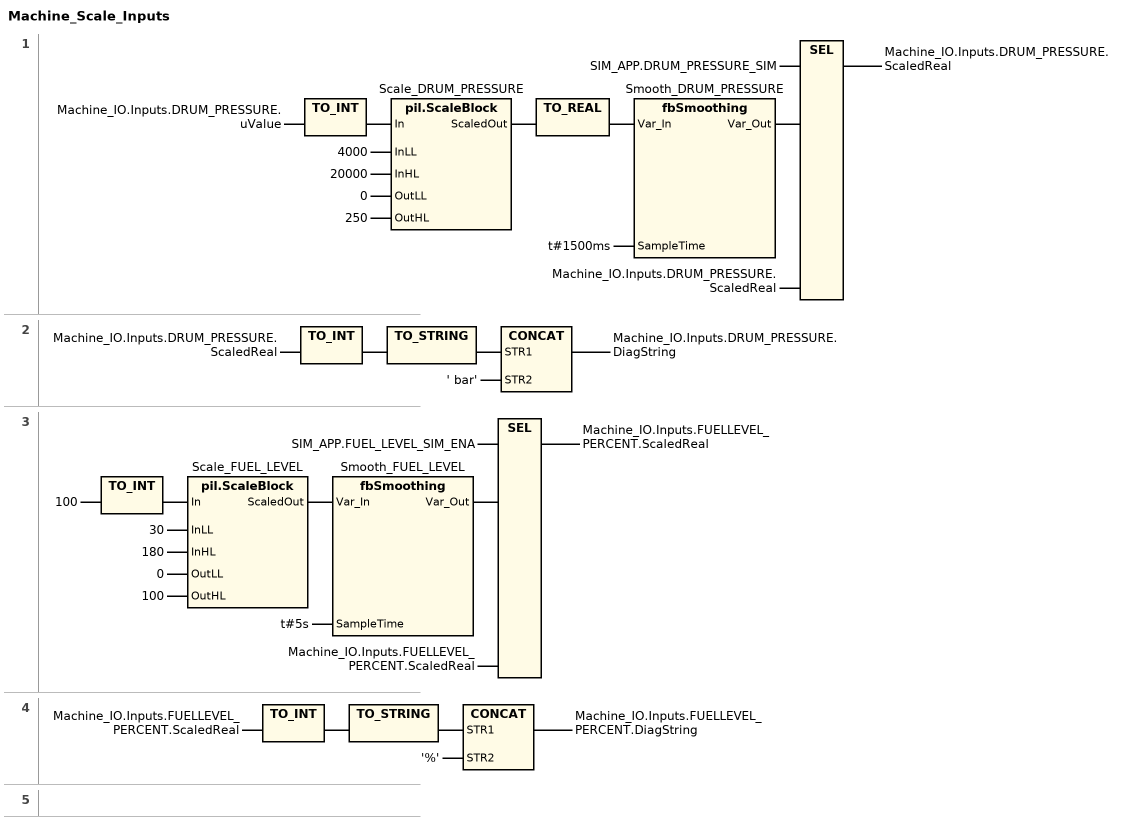
// NETWORK 1
Scale_DRUM_PRESSURE(
    In := TO_INT(Machine_IO.Inputs.DRUM_PRESSURE.uValue),
    InLL := 4000,
    InHL := 20000,
    OutLL := 0,
    OutHL := 250); // pil.ScaleBlock
Smooth_DRUM_PRESSURE(Var_In := TO_REAL(Scale_DRUM_PRESSURE.ScaledOut), SampleTime := t#1500ms); // fbSmoothing
Machine_IO.Inputs.DRUM_PRESSURE.ScaledReal := SEL(SIM_APP.DRUM_PRESSURE_SIM, Smooth_DRUM_PRESSURE.Var_Out, Machine_IO.Inputs.DRUM_PRESSURE.ScaledReal);

// NETWORK 2
Machine_IO.Inputs.DRUM_PRESSURE.DiagString := CONCAT(STR1 := TO_STRING(TO_INT(Machine_IO.Inputs.DRUM_PRESSURE.ScaledReal)), STR2 := ' bar');

// NETWORK 3
Scale_FUEL_LEVEL(In := TO_INT(100), InLL := 30, InHL := 180, OutLL := 0, OutHL := 100); // pil.ScaleBlock
Smooth_FUEL_LEVEL(Var_In := Scale_FUEL_LEVEL.ScaledOut, SampleTime := t#5s); // fbSmoothing
Machine_IO.Inputs.FUELLEVEL_PERCENT.ScaledReal := SEL(SIM_APP.FUEL_LEVEL_SIM_ENA, Smooth_FUEL_LEVEL.Var_Out, Machine_IO.Inputs.FUELLEVEL_PERCENT.ScaledReal);

// NETWORK 4
Machine_IO.Inputs.FUELLEVEL_PERCENT.DiagString := CONCAT(STR1 := TO_STRING(TO_INT(Machine_IO.Inputs.FUELLEVEL_PERCENT.ScaledReal)), STR2 := '%');

// NETWORK 5

END_PROGRAM

// Device/Application/App_PLC/fbSmoothing
FUNCTION_BLOCK fbSmoothing
VAR_INPUT
	Var_In: REAL;
	SampleTime: TIME;
END_VAR
VAR_OUTPUT
	Var_Out: REAL;
END_VAR
VAR
	Timer: TON;
	SampleArray: ARRAY [0..49] OF REAL;
	ArraySampleTime: TIME;
	Timer2: TON;
END_VAR

ArraySampleTime:= SampleTime/50;
Timer(IN:=NOT Timer.Q, PT:=ArraySampleTime, Q=>, ET=> );

IF Timer.Q=TRUE THEN

SampleArray[49]:=SampleArray[48];
SampleArray[48]:=SampleArray[47];
SampleArray[47]:=SampleArray[46];
SampleArray[46]:=SampleArray[45];
SampleArray[45]:=SampleArray[44];
SampleArray[44]:=SampleArray[43];
SampleArray[43]:=SampleArray[42];
SampleArray[42]:=SampleArray[41];
SampleArray[41]:=SampleArray[40];
SampleArray[40]:=SampleArray[39];
SampleArray[39]:=SampleArray[38];
SampleArray[38]:=SampleArray[37];
SampleArray[37]:=SampleArray[36];
SampleArray[36]:=SampleArray[35];
SampleArray[35]:=SampleArray[34];
SampleArray[34]:=SampleArray[33];
SampleArray[33]:=SampleArray[32];
SampleArray[32]:=SampleArray[31];
SampleArray[31]:=SampleArray[30];
SampleArray[30]:=SampleArray[29];
SampleArray[29]:=SampleArray[28];
SampleArray[28]:=SampleArray[27];
SampleArray[27]:=SampleArray[26];
SampleArray[26]:=SampleArray[25];
SampleArray[25]:=SampleArray[24];
SampleArray[24]:=SampleArray[23];
SampleArray[23]:=SampleArray[22];
SampleArray[22]:=SampleArray[21];
SampleArray[21]:=SampleArray[20];
SampleArray[20]:=SampleArray[19];
SampleArray[19]:=SampleArray[18];
SampleArray[18]:=SampleArray[17];
SampleArray[17]:=SampleArray[16];
SampleArray[16]:=SampleArray[15];
SampleArray[15]:=SampleArray[14];
SampleArray[14]:=SampleArray[13];
SampleArray[13]:=SampleArray[12];
SampleArray[12]:=SampleArray[11];
SampleArray[11]:=SampleArray[10];
SampleArray[10]:=SampleArray[9];
SampleArray[9]:=SampleArray[8];
SampleArray[8]:=SampleArray[7];
SampleArray[7]:=SampleArray[6];
SampleArray[6]:=SampleArray[5];
SampleArray[5]:=SampleArray[4];
SampleArray[4]:=SampleArray[3];
SampleArray[3]:=SampleArray[2];
SampleArray[2]:=SampleArray[1];
SampleArray[1]:=SampleArray[0];
SampleArray[0]:=Var_In;
END_IF

Timer2(IN:=NOT Timer2.Q, PT:=SampleTime, Q=>, ET=> );

IF Timer2.Q=TRUE THEN
Var_Out:= (
SampleArray[49] + SampleArray[48] + SampleArray[47] + SampleArray[46] + SampleArray[45] + SampleArray[44] + SampleArray[43] + SampleArray[42] + SampleArray[41] +SampleArray[40] +
SampleArray[39] + SampleArray[38] + SampleArray[37] + SampleArray[36] + SampleArray[35] + SampleArray[34] + SampleArray[33] + SampleArray[32] + SampleArray[31] +SampleArray[30] +
SampleArray[29] + SampleArray[28] + SampleArray[27] + SampleArray[26] + SampleArray[25] + SampleArray[24] + SampleArray[23] + SampleArray[22] + SampleArray[21] +SampleArray[20] +
SampleArray[19] + SampleArray[18] + SampleArray[17] + SampleArray[16] + SampleArray[15] + SampleArray[14] + SampleArray[13] + SampleArray[12] + SampleArray[11] +SampleArray[10] +
SampleArray[9] + SampleArray[8] + SampleArray[7] + SampleArray[6] + SampleArray[5] + SampleArray[4] + SampleArray[3] + SampleArray[2] + SampleArray[1] +SampleArray[0]
			)/50;
END_IF

END_FUNCTION_BLOCK

// Device/Application/LIBS/Logging/Log_File_Append
FUNCTION Log_File_Append : INT
VAR_INPUT
	LogString: STRING;
	szFileName : STRING;		
	Updated_Flag: REFERENCE TO INT;
END_VAR
VAR	
	hFile : RTS_IEC_HANDLE := RTS_INVALID_HANDLE;
	
	udiWriteError : RTS_IEC_RESULT;
	udiOpenError : RTS_IEC_RESULT;
	udiCloseError : RTS_IEC_RESULT;
	udiWrite : __XWORD;
	
	TempString: STRING;
	
	High_Res_millis: INT:=0;
	High_Res_Timestamp:	SYSTIME;
	High_Res_Timestamp_Result: RTS_IEC_RESULT;
	High_Res_Timestamp_DT: DT;
	High_Res_Timestamp_String: STRING;
END_VAR

// get the high res time stamp that has milliseconds
High_Res_Timestamp_Result:=SysTimeRtc.SysTimeRtcHighResGet(High_Res_Timestamp);

IF High_Res_Timestamp_Result <> CmpErrors.Errors.ERR_OK THEN
	Log_File_Append:=-1;
	RETURN;	
END_IF

High_Res_Timestamp_DT := TO_DT(High_Res_Timestamp/1000);
High_Res_millis := TO_INT(High_Res_Timestamp MOD 1000);

High_Res_Timestamp_String := OSCAT_BASIC.DT_TO_STRF(DTI:=High_Res_Timestamp_DT, MS:=High_Res_millis, FMT:='#N:#R:#T.#V,#H-#D-#A',LANG:=OSCAT_BASIC.language.DEFAULT);

hFile := SysFileOpen(szFile:=szFileName, am:=SysFile.AM_APPEND_PLUS, pResult:=ADR(udiOpenError));

IF hFile <> RTS_INVALID_HANDLE	THEN
	TempString:=CONCAT(TempString,LogString);	
	TempString:=CONCAT(TempString,',');
	TempString:=CONCAT(TempString,High_Res_Timestamp_String);	
	TempString:=CONCAT(TempString,'$0d$0a');
	udiWrite := SysFileWrite(hFile:=hFile, pbyBuffer:=ADR(TempString), ulSize:=INT_TO_UDINT(LEN(TempString)), pResult:=ADR(udiWriteError));

	udiCloseError  := SysFileClose(hFile:=hFile);
	Log_File_Append:=0;
	Updated_Flag:=Updated_Flag+1;
	RETURN;
END_IF

Log_File_Append:=-2;
RETURN;

END_FUNCTION

// Device/Application/App_Common/System/PLC_LOGGING
PROGRAM PLC_LOGGING
VAR
	Main_Log_Update: BOOL;
	Main_Log_Update_Reset_TON: TON;
	
	LOG_LINES: ARRAY [0..9] OF STRING(200);
	Log_File_Read_Lines_Check_FB: Log_File_Read_Lines;
	Log_File_Read_Lines_FB: Log_File_Read_Lines;
	MaxLines: INT :=10;
	
	Offset: INT;
	Number_Lines: INT;
END_VAR
VAR // added by the converter: edge detectors and wires of the graphical bodies
    _rt1, _rt2, _rt3, _rt4, _rt5 : R_TRIG;
    _w1, _w2, _w3 : BOOL;
END_VAR

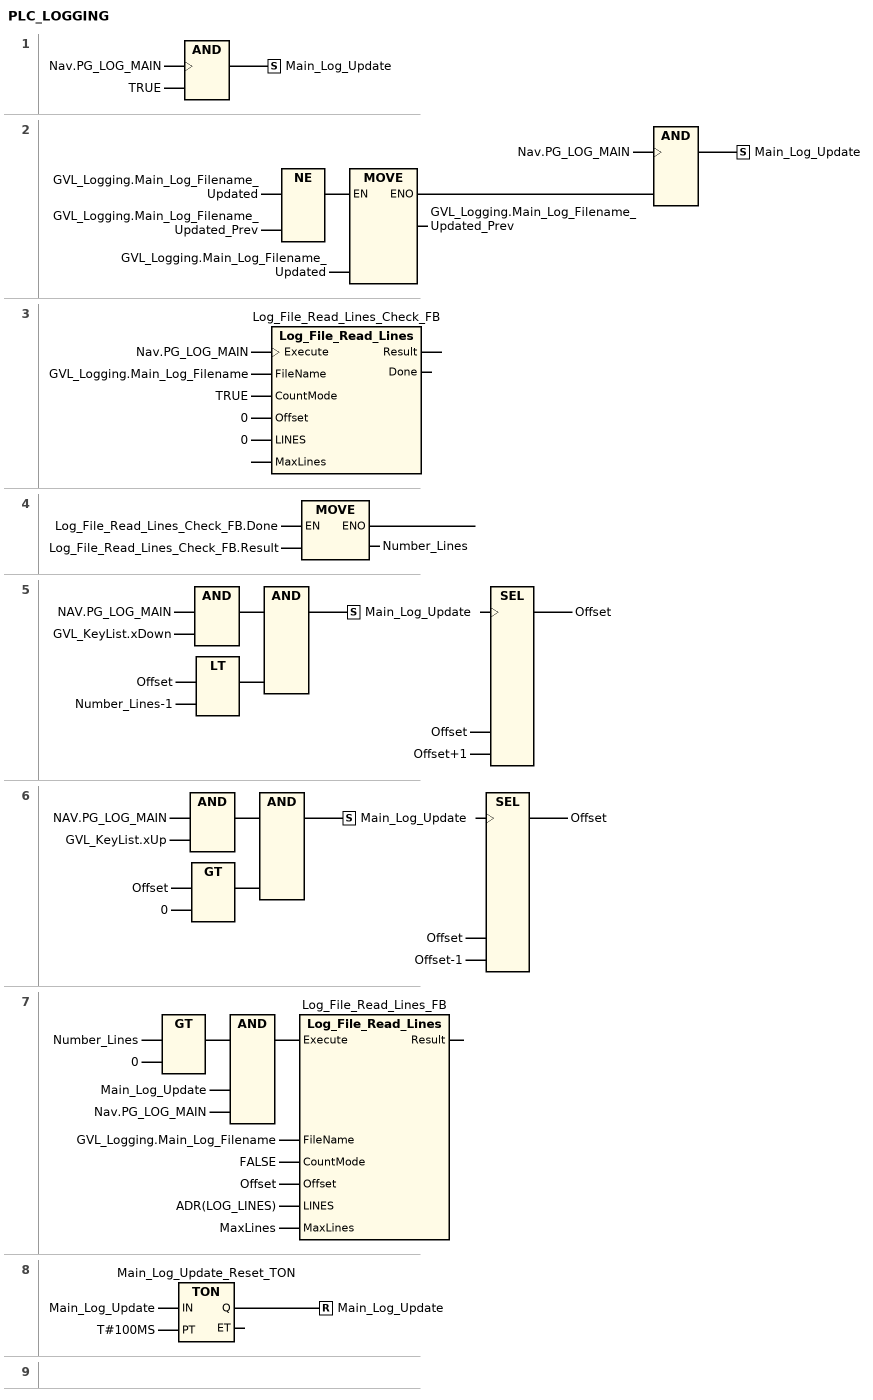
// NETWORK 1
_rt1(CLK := Nav.PG_LOG_MAIN);
Main_Log_Update S= _rt1.Q AND TRUE;

// NETWORK 2
_rt2(CLK := Nav.PG_LOG_MAIN);
_w1 := GVL_Logging.Main_Log_Filename_Updated <> GVL_Logging.Main_Log_Filename_Updated_Prev;
IF _w1 THEN GVL_Logging.Main_Log_Filename_Updated_Prev := GVL_Logging.Main_Log_Filename_Updated; END_IF
Main_Log_Update S= _rt2.Q AND _w1;

// NETWORK 3
_rt3(CLK := Nav.PG_LOG_MAIN);
Log_File_Read_Lines_Check_FB(
    Execute := _rt3.Q,
    FileName := GVL_Logging.Main_Log_Filename,
    CountMode := TRUE,
    Offset := 0,
    LINES := 0); // Log_File_Read_Lines

// NETWORK 4
IF Log_File_Read_Lines_Check_FB.Done THEN Number_Lines := Log_File_Read_Lines_Check_FB.Result; END_IF

// NETWORK 5
_w2 := (NAV.PG_LOG_MAIN AND GVL_KeyList.xDown) AND Offset < (Number_Lines-1);
Main_Log_Update S= _w2;
_rt4(CLK := _w2);
Offset := SEL(_rt4.Q, Offset, Offset+1);

// NETWORK 6
_w3 := (NAV.PG_LOG_MAIN AND GVL_KeyList.xUp) AND Offset > 0;
Main_Log_Update S= _w3;
_rt5(CLK := _w3);
Offset := SEL(_rt5.Q, Offset, Offset-1);

// NETWORK 7
Log_File_Read_Lines_FB(
    Execute := Number_Lines > 0 AND Main_Log_Update AND Nav.PG_LOG_MAIN,
    FileName := GVL_Logging.Main_Log_Filename,
    CountMode := FALSE,
    Offset := Offset,
    LINES := ADR(LOG_LINES),
    MaxLines := MaxLines); // Log_File_Read_Lines

// NETWORK 8
Main_Log_Update_Reset_TON(IN := Main_Log_Update, PT := T#100MS); // TON
Main_Log_Update R= Main_Log_Update_Reset_TON.Q;

// NETWORK 9

END_PROGRAM

// Device/Application/LIBS/Logging/Log_File_Read_Lines
FUNCTION_BLOCK Log_File_Read_Lines
VAR_INPUT
	Execute: BOOL;
	FileName: STRING;
	CountMode: BOOL;
	Offset: INT:=0;
	LINES: POINTER TO STRING(200);	
	MaxLines: INT:=10;
END_VAR
VAR	
	hFile : RTS_IEC_HANDLE := RTS_INVALID_HANDLE;
	
	udiReadError : RTS_IEC_RESULT;
	udiOpenError : RTS_IEC_RESULT;
	udiCloseError : RTS_IEC_RESULT;
	udiWrite : __XWORD;
	ReadSize : __XWORD;
	
	TempString: STRING(2);
	LineBuffer: STRING(200);
	
	NumLines:INT:=0;
	line_counter:INT :=0;

	op_index:INT :=0;
	dummy: INT;
	Finished:BOOL:=FALSE;
END_VAR

VAR_OUTPUT
	Result:INT;
	Done: BOOL;
END_VAR

IF Execute = FALSE THEN
	Result:=0;
	Done:=0;
	RETURN;
END_IF

IF MaxLines = 0 THEN
	RETURN;
END_IF

IF LINES <> 0 THEN
	FOR line_counter := 0 TO (MaxLines-1) BY 1 DO
		LINES[line_counter]:='';
	END_FOR;	
END_IF

IF CountMode = FALSE AND LINES = 0 THEN
	Result:= -1;
	RETURN;
END_IF

hFile := SysFileOpen(szFile:=FileName, am:=SysFile.AM_READ, pResult:=ADR(udiOpenError));

IF hFile = RTS_INVALID_HANDLE THEN
	Result:=-2;
	RETURN;	
END_IF

Finished := FALSE;

line_counter:=0;
LineBuffer:='';

WHILE Finished = FALSE DO
	ReadSize := SysFileRead(hFile:=hFile, pbyBuffer:=ADR(TempString), ulSize:=1, pResult:=ADR(udiReadError));
	
	IF ReadSize<= 0 THEN
		Finished:=TRUE;
	END_IF
	
	TempString:=LEFT(TempString,1);
	IF(TempString='$0D') THEN
		op_index:=line_counter-Offset;	
		IF op_index >= 0 AND op_index < (MaxLines-1) THEN
			IF CountMode = FALSE AND op_index < MaxLines AND (LEN(LineBuffer)>0) THEN
				IF LINES <> 0 THEN
					LINES[op_index]:='[';
					LINES[op_index]:=CONCAT(LINES[op_index],TO_STRING(line_counter));
					LINES[op_index]:=CONCAT(LINES[op_index],'] ');
					LINES[op_index]:=CONCAT(LINES[op_index],LineBuffer);				
				END_IF
			END_IF			
		END_IF
		line_counter:=line_counter+1;		
		LineBuffer:='';		
		
	ELSIF(TempString='$0A') THEN
		dummy:=dummy+1;
	ELSE
		LineBuffer:=CONCAT(LineBuffer,TempString);
	END_IF
END_WHILE

udiCloseError  := SysFileClose(hFile:=hFile);
Result:=line_counter;
Done:=1;
RETURN;

END_FUNCTION_BLOCK

// Device/Application/LIBS/Alarms/Functions/Alarm_Table_Main
PROGRAM Alarm_Table_Main
VAR CONSTANT
	NUM_LINES: WORD:=5;
END_VAR

VAR
	BASE_INDEX:WORD:=0;
	Lines: ARRAY [0..(NUM_LINES-1)] OF Alarm_Logger_Line_FB;
	INDEXS: ARRAY [0..(NUM_LINES-1)] OF WORD;
	X:WORD;
END_VAR

VAR_INPUT
	LIST: REFERENCE TO SLL_LOGGER_MAIN_SRUCT;
	NAV_UP: BOOL;
	NAV_DOWN: BOOL;
END_VAR


FOR X:= 0 TO (NUM_LINES-1) DO
	INDEXS[X]:=(BASE_INDEX+X) MOD LIST.LOGGER_LIST_SIZE;	
	Lines[X](INDEX:=INDEXS[X],ITEM:=LIST.LOGGER_LIST[INDEXS[X]]);
END_FOR

IF NAV_UP THEN
	IF BASE_INDEX > 0 THEN 
		BASE_INDEX:=BASE_INDEX-1;
	ELSE
		BASE_INDEX:= LIST.LOGGER_LIST_SIZE-1;
	END_IF
END_IF

IF NAV_DOWN THEN
	IF BASE_INDEX <  (LIST.LOGGER_LIST_SIZE-2) THEN 
		BASE_INDEX:=BASE_INDEX+1;
	ELSE
		BASE_INDEX:= 0;
	END_IF
END_IF

END_PROGRAM

// Device/Application/LIBS/Alarms/Functions/Alarm_Logger_Line_FB
FUNCTION_BLOCK Alarm_Logger_Line_FB
VAR_INPUT
	INDEX: WORD;
	ITEM: REFERENCE TO SLL_LOGGER_ITEM;
END_VAR
VAR_OUTPUT
	oIndex:STRING;
	oID:STRING;
	oDescription: STRING;
	oTime: STRING;
	oAdd_Info: STRING;
	oSquareColour: DWORD;
END_VAR
VAR
	InitDone:BOOL :=FALSE;
	TempString: STRING;
	
	High_Res_millis: INT:=0;
	High_Res_Timestamp:	SYSTIME;
	High_Res_Timestamp_DT: DT;
END_VAR


oIndex:='[';
oIndex:=CONCAT(oIndex,TO_STRING(INDEX));
oIndex:=CONCAT(oIndex,']');

IF ITEM.ID > 0 THEN
	oID:=CONCAT('ID:',TO_STRING(ITEM.ID));	
	IF ITEM.Group.ErrorIO OR ITEM.Group.WarningIO THEN
		TempString := Alarm_ID_GetText('AlarmGroup_IO',TO_STRING(ITEM.ID));
	END_IF

	IF ITEM.Group.ErrorApp OR ITEM.Group.WarningApp THEN
		TempString := Alarm_ID_GetText('AlarmGroup_App',TO_STRING(ITEM.ID));
	END_IF
		

	IF TempString = '' THEN
		oDescription:=TO_STRING(ITEM.ID);
	END_IF;
	
	oDescription:=TempString;
	
	High_Res_Timestamp:=ITEM.TimeDateTriggered;
	High_Res_Timestamp_DT := TO_DT(High_Res_Timestamp/1000);
	High_Res_millis := TO_INT(High_Res_Timestamp MOD 1000);
	IF GVL_System.USA_Time_Format THEN
		oTime:= OSCAT_BASIC.DT_TO_STRF(DTI:=High_Res_Timestamp_DT, MS:=High_Res_millis, FMT:='#N:#R:#T.#V,#D-#H-#A',LANG:=OSCAT_BASIC.language.DEFAULT);
	ELSE
		oTime:= OSCAT_BASIC.DT_TO_STRF(DTI:=High_Res_Timestamp_DT, MS:=High_Res_millis, FMT:='#N:#R:#T.#V,#H-#D-#A',LANG:=OSCAT_BASIC.language.DEFAULT);
	END_IF

	oAdd_Info:=ITEM.Addtional_Info;
	
	IF ITEM.Flags.Active THEN
		oSquareColour:=GVL_Viz.Alarm_Log_Active_Colour;
	ELSE
		oSquareColour:=GVL_Viz.Alarm_Log_InActive_Colour;
	END_IF
ELSE
	oID:='';
	oDescription:='';
	oTime:='';
	oAdd_Info:='';
	oSquareColour:=GVL_Viz.Alarm_Log_None_Colour;
END_IF

END_FUNCTION_BLOCK

// Device/Application/LIBS/Alarms/Functions/Alarm_ID_GetText
FUNCTION Alarm_ID_GetText : STRING
VAR_INPUT
	TextListName: STRING;
	ItemName:STRING;	
END_VAR
VAR
	Current : STRING:='';
	TextListItem:STRING:='';
END_VAR

Current := DynamicTextGetCurrentLanguage();

IF Current = '' THEN
	TextListItem:=DynamicTextGetDefaultText(ADR(TextListName), ADR(ItemName))^;
ELSE
	TextListItem:=DynamicTextGetText(ADR(TextListName), ADR(ItemName))^;
END_IF

Alarm_ID_GetText:=TextListItem;

END_FUNCTION

// Device/Application/LIBS/Alarms/Functions/Alarm_Log_Clear_ALL
FUNCTION Alarm_Log_Clear_ALL : INT
VAR_INPUT
	LIST: REFERENCE TO SLL_LOGGER_MAIN_SRUCT;
	ENA: BOOL;
END_VAR
VAR_OUTPUT
END_VAR
VAR
	X:WORD;
	Empty_ITEM:SLL_LOGGER_ITEM;
END_VAR

IF ENA = FALSE THEN
	RETURN;	
END_IF

FOR X :=0 TO (LIST.LOGGER_LIST_SIZE-1) BY 1 DO
	LIST.LOGGER_LIST[X]:=Empty_ITEM;
END_FOR

END_FUNCTION

// Device/Application/LIBS/Alarms/Functions/Alarm_Log_Clear_ALL_Inactive
FUNCTION Alarm_Log_Clear_ALL_Inactive : INT
VAR_INPUT
	LIST: REFERENCE TO SLL_LOGGER_MAIN_SRUCT;
	ENA: BOOL;
END_VAR
VAR_OUTPUT
END_VAR
VAR
	X:WORD;
	Z:WORD;
	Empty_ITEM:SLL_LOGGER_ITEM;
END_VAR

IF ENA = FALSE THEN
	RETURN;	
END_IF

FOR X :=0 TO (LIST.LOGGER_LIST_SIZE-1) BY 1 DO
	IF LIST.LOGGER_LIST[X].ID > 0 THEN
		// got a id of some sort...
		IF LIST.LOGGER_LIST[X].Flags.Active = FALSE THEN
			// wipe this record 
			LIST.LOGGER_LIST[X]:=Empty_ITEM;
	
			// loose this record..shift up the date towards the start!
			FOR Z:= X TO (LIST.LOGGER_LIST_SIZE-2) BY 1 DO
				LIST.LOGGER_LIST[Z]:=LIST.LOGGER_LIST[Z+1];
			END_FOR
			
			// clear the last record since we got rid of one!
			LIST.LOGGER_LIST[Z]:=Empty_ITEM;
			
			IF X>0 THEN
				X:=X-1; // we need to re-run this loop!
			END_IF;
		END_IF	
	END_IF
END_FOR

END_FUNCTION

// Device/Application/App_Common/Nav/Page Control/LED_Ctrl
PROGRAM LED_Ctrl
VAR
	F1_LED_ON: ifmDevice.SetKeyLED;
	F1_LED_OFF: ifmDevice.SetKeyLED;
	F2_LED_ON: ifmDevice.SetKeyLED;
	F2_LED_OFF: ifmDevice.SetKeyLED;
	F3_LED_ON: ifmDevice.SetKeyLED;
	F3_LED_OFF: ifmDevice.SetKeyLED;
	F4_LED_ON: ifmDevice.SetKeyLED;
	F4_LED_OFF: ifmDevice.SetKeyLED;
	F5_LED_ON: ifmDevice.SetKeyLED;
	F5_LED_OFF: ifmDevice.SetKeyLED;
	F6_LED_ON: ifmDevice.SetKeyLED;
	F6_LED_OFF: ifmDevice.SetKeyLED;
	NavKey_LED_ON: ifmDevice.SetKeyLED;
	NavKey_LED_OFF: ifmDevice.SetKeyLED;
END_VAR

VAR_INPUT
	F1_On: BOOL;
	F1_Colour:DWORD:=16#00994C00;
	F2_On: BOOL;
	F2_Colour:DWORD:=16#00994C00;
	F3_On: BOOL;
	F3_Colour:DWORD:=16#00994C00;
	F4_On: BOOL;
	F4_Colour:DWORD:=16#00994C00;
	F5_On: BOOL;
	F5_Colour:DWORD:=16#00994C00;
 	F6_On: BOOL;
	F6_Colour:DWORD:=16#00FFFFFF;
	Nav_On: BOOL;
	Nav_Colour: DWORD:=16#0000FF00;
END_VAR

F1_LED_ON (xEnable:=F1_On, eLED_ID:=16#0, udiColour:=F1_Colour, stNightMode:=,  xError=>, eDiagInfo=>);
F1_LED_OFF (xEnable:=NOT F1_On, eLED_ID:=16#0, udiColour:=16#00000000, stNightMode:=,  xError=>, eDiagInfo=>);

F2_LED_ON (xEnable:=F2_On, eLED_ID:=16#1, udiColour:=F2_Colour, stNightMode:=,  xError=>, eDiagInfo=>);
F2_LED_OFF (xEnable:=NOT F2_On, eLED_ID:=16#1, udiColour:=16#00000000, stNightMode:=,  xError=>, eDiagInfo=>);

F3_LED_ON (xEnable:=F3_On, eLED_ID:=16#2, udiColour:=F3_Colour, stNightMode:=,  xError=>, eDiagInfo=>);
F3_LED_OFF (xEnable:=NOT F3_On, eLED_ID:=16#2, udiColour:=16#00000000, stNightMode:=,  xError=>, eDiagInfo=>);

F4_LED_ON (xEnable:=F4_On, eLED_ID:=16#3, udiColour:=F4_Colour, stNightMode:=,  xError=>, eDiagInfo=>);
F4_LED_OFF (xEnable:=NOT F4_On, eLED_ID:=16#3, udiColour:=16#00000000, stNightMode:=,  xError=>, eDiagInfo=>);

F5_LED_ON (xEnable:=F5_On, eLED_ID:=16#4, udiColour:=F5_Colour, stNightMode:=,  xError=>, eDiagInfo=>);
F5_LED_OFF (xEnable:=NOT F5_On, eLED_ID:=16#4, udiColour:=16#00000000, stNightMode:=,  xError=>, eDiagInfo=>);

F6_LED_ON (xEnable:=F6_On, eLED_ID:=16#5, udiColour:=F6_Colour, stNightMode:=,  xError=>, eDiagInfo=>);
F6_LED_OFF (xEnable:=NOT F6_On, eLED_ID:=16#5, udiColour:=16#00000000, stNightMode:=,  xError=>, eDiagInfo=>);

NavKey_LED_ON (xEnable:=NAV_On, eLED_ID:=16#B, udiColour:=Nav_Colour, stNightMode:=,  xError=>, eDiagInfo=>);
NavKey_LED_OFF (xEnable:=NOT Nav_On, eLED_ID:=16#B, udiColour:=16#00000000, stNightMode:=,  xError=>, eDiagInfo=>);

END_PROGRAM

// Device/Application/App_Common/Nav/Page Control/LED_Control_FB
FUNCTION_BLOCK LED_Control_FB
VAR	
	F1_LED_ON: ifmDevice.SetKeyLED;
	F1_LED_OFF: ifmDevice.SetKeyLED;
	F2_LED_ON: ifmDevice.SetKeyLED;
	F2_LED_OFF: ifmDevice.SetKeyLED;
	F3_LED_ON: ifmDevice.SetKeyLED;
	F3_LED_OFF: ifmDevice.SetKeyLED;
	F4_LED_ON: ifmDevice.SetKeyLED;
	F4_LED_OFF: ifmDevice.SetKeyLED;
	F5_LED_ON: ifmDevice.SetKeyLED;
	F5_LED_OFF: ifmDevice.SetKeyLED;
	F6_LED_ON: ifmDevice.SetKeyLED;
	F6_LED_OFF: ifmDevice.SetKeyLED;
	NavKey_LED_ON: ifmDevice.SetKeyLED;
	NavKey_LED_OFF: ifmDevice.SetKeyLED;
	Dummy_LED_ON: ifmDevice.SetKeyLED;
	Dummy_LED_OFF: ifmDevice.SetKeyLED;
	Dummy_State: BOOL;
	Ena_Prev: BOOL;
	COUNTER:WORD;
END_VAR

VAR_INPUT
	Ena: BOOL;
	F1_On: BOOL;
	F1_Colour:DWORD:=16#00994C00;
	F2_On: BOOL;
	F2_Colour:DWORD:=16#00994C00;
	F3_On: BOOL;
	F3_Colour:DWORD:=16#00994C00;
	F4_On: BOOL;
	F4_Colour:DWORD:=16#00994C00;
	F5_On: BOOL;
	F5_Colour:DWORD:=16#00994C00;
 	Home_On: BOOL;
	Home_Colour:DWORD:=16#00994C00;
	Nav_On: BOOL;
	Nav_Colour: DWORD:=16#0000FF00;	
END_VAR
VAR_OUTPUT
END_VAR
VAR
END_VAR

IF Ena = TRUE THEN
	IF COUNTER < 10 THEN
		COUNTER:=COUNTER+1;
		RETURN;
	END_IF
	// run the code below!
ELSE
	Ena_Prev:=FALSE;
	COUNTER:=0;
	RETURN;
END_IF

Dummy_State:=NOT Dummy_State;

F1_LED_ON (xEnable:=F1_On, eLED_ID:=16#4, udiColour:=F1_Colour, stNightMode:=,  xError=>, eDiagInfo=>);
F1_LED_OFF (xEnable:=NOT F1_On, eLED_ID:=16#4, udiColour:=16#00000000, stNightMode:=,  xError=>, eDiagInfo=>);

F2_LED_ON (xEnable:=F2_On, eLED_ID:=16#2, udiColour:=F2_Colour, stNightMode:=,  xError=>, eDiagInfo=>);
F2_LED_OFF (xEnable:=NOT F2_On, eLED_ID:=16#2, udiColour:=16#00000000, stNightMode:=,  xError=>, eDiagInfo=>);

F3_LED_ON (xEnable:=F3_On, eLED_ID:=16#0, udiColour:=F3_Colour, stNightMode:=,  xError=>, eDiagInfo=>);
F3_LED_OFF (xEnable:=NOT F3_On, eLED_ID:=16#0, udiColour:=16#00000000, stNightMode:=,  xError=>, eDiagInfo=>);

F4_LED_ON (xEnable:=F4_On, eLED_ID:=16#1, udiColour:=F4_Colour, stNightMode:=,  xError=>, eDiagInfo=>);
F4_LED_OFF (xEnable:=NOT F4_On, eLED_ID:=16#1, udiColour:=16#00000000, stNightMode:=,  xError=>, eDiagInfo=>);

F5_LED_ON (xEnable:=F5_On, eLED_ID:=16#3, udiColour:=F5_Colour, stNightMode:=,  xError=>, eDiagInfo=>);
F5_LED_OFF (xEnable:=NOT F5_On, eLED_ID:=16#3, udiColour:=16#00000000, stNightMode:=,  xError=>, eDiagInfo=>);

F6_LED_ON (xEnable:=Home_On, eLED_ID:=16#5, udiColour:=Home_Colour, stNightMode:=,  xError=>, eDiagInfo=>);
F6_LED_OFF (xEnable:=NOT Home_On, eLED_ID:=16#5, udiColour:=16#00000000, stNightMode:=,  xError=>, eDiagInfo=>);

F6_LED_ON (xEnable:=Home_On, eLED_ID:=16#5, udiColour:=Home_Colour, stNightMode:=,  xError=>, eDiagInfo=>);
F6_LED_OFF (xEnable:=NOT Home_On, eLED_ID:=16#5, udiColour:=16#00000000, stNightMode:=,  xError=>, eDiagInfo=>);

// DUMMY_LED_ON (xEnable:=Dummy_State,eLED_ID:=16#6, udiColour:=16#00FFFFFF, stNightMode:=,  xError=>, eDiagInfo=>);
// DUMMY_LED_OFF (xEnable:=NOT Dummy_State,eLED_ID:=16#6, udiColour:=16#00000000, stNightMode:=,  xError=>, eDiagInfo=>);

NavKey_LED_ON (xEnable:=NAV_On, eLED_ID:=16#B, udiColour:=Nav_Colour, stNightMode:=,  xError=>, eDiagInfo=>);
NavKey_LED_OFF (xEnable:=NOT Nav_On, eLED_ID:=16#B, udiColour:=16#00000000, stNightMode:=,  xError=>, eDiagInfo=>);

END_FUNCTION_BLOCK

// Device/Application/App_Common/System/PLC_GET_SET_IP_ADDRESS
PROGRAM PLC_GET_SET_IP_ADDRESS
VAR
	GET_IP_SETTINGS: BOOL:=TRUE;
// 	GetIPSettings_FB: ifmDevice.GetIPsettings2;
// 	Get_IP_Setup: ifmDevice.stIP_SETTING;
// 
// 	SetIPSettings_FB: ifmDevice.SetIPsettings2;
	SET_IP_SETTINGS: BOOL;
// 	IP_Setup: ifmDevice.stIP_SETTING;
	
	IP_LOCAL_ADDRESS: STRING := '192.168.82.245';
	IP_LOCAL_GATEWAY: STRING := '192.168.82.1';	
	ShutdownDevice_FB: ifmDevice.ShutdownDevice;
	DONE: BOOL;
	SET_IP_SETTINGS_TON: TON;
END_VAR
VAR // added by the converter: edge detectors and wires of the graphical bodies
    _rt1, _rt2 : R_TRIG;
END_VAR

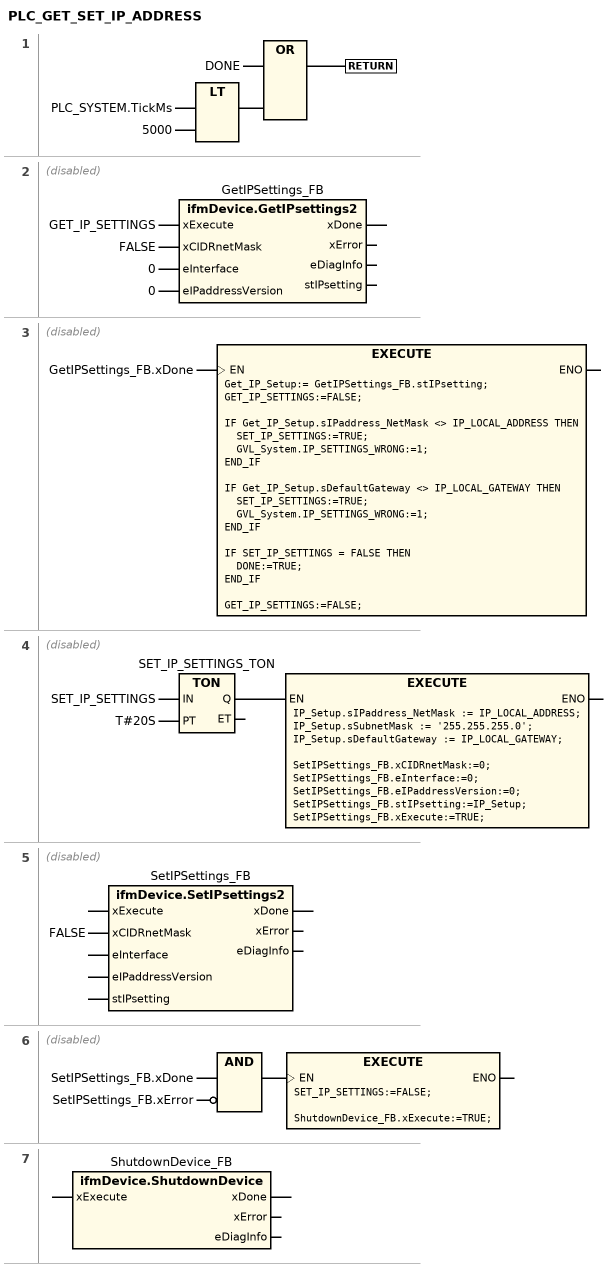
// NETWORK 1
IF DONE OR PLC_SYSTEM.TickMs < 5000 THEN RETURN; END_IF

// NETWORK 2 (disabled)
// GetIPSettings_FB(xExecute := GET_IP_SETTINGS, xCIDRnetMask := FALSE, eInterface := 0, eIPaddressVersion := 0); // ifmDevice.GetIPsettings2

// NETWORK 3 (disabled)
// _rt1(CLK := GetIPSettings_FB.xDone);
// IF _rt1.Q THEN
//     Get_IP_Setup:= GetIPSettings_FB.stIPsetting;
//     GET_IP_SETTINGS:=FALSE;
//     
//     IF Get_IP_Setup.sIPaddress_NetMask <> IP_LOCAL_ADDRESS THEN
//     	SET_IP_SETTINGS:=TRUE;
//     	GVL_System.IP_SETTINGS_WRONG:=1;
//     END_IF
//     
//     IF Get_IP_Setup.sDefaultGateway <> IP_LOCAL_GATEWAY THEN
//     	SET_IP_SETTINGS:=TRUE;
//     	GVL_System.IP_SETTINGS_WRONG:=1;
//     END_IF
//     
//     IF SET_IP_SETTINGS = FALSE THEN
//     	DONE:=TRUE;
//     END_IF
//     
//     GET_IP_SETTINGS:=FALSE;
// END_IF

// NETWORK 4 (disabled)
// SET_IP_SETTINGS_TON(IN := SET_IP_SETTINGS, PT := T#20S); // TON
// IF SET_IP_SETTINGS_TON.Q THEN
//     IP_Setup.sIPaddress_NetMask := IP_LOCAL_ADDRESS;
//     IP_Setup.sSubnetMask := '255.255.255.0';
//     IP_Setup.sDefaultGateway := IP_LOCAL_GATEWAY;
//     
//     SetIPSettings_FB.xCIDRnetMask:=0;
//     SetIPSettings_FB.eInterface:=0;
//     SetIPSettings_FB.eIPaddressVersion:=0;
//     SetIPSettings_FB.stIPsetting:=IP_Setup;
//     SetIPSettings_FB.xExecute:=TRUE;
// END_IF

// NETWORK 5 (disabled)
// SetIPSettings_FB(xCIDRnetMask := FALSE); // ifmDevice.SetIPsettings2

// NETWORK 6 (disabled)
// _rt2(CLK := SetIPSettings_FB.xDone AND NOT SetIPSettings_FB.xError);
// IF _rt2.Q THEN
//     SET_IP_SETTINGS:=FALSE;
//     
//     ShutdownDevice_FB.xExecute:=TRUE;
// END_IF

// NETWORK 7
ShutdownDevice_FB(); // ifmDevice.ShutdownDevice

END_PROGRAM

// Device/Application/App_Common/Machine/Safety_Common
PROGRAM Safety_Common
VAR
	Estop_Signal_DB: SWITCH_DEBOUNCE;
	ESTOP_OK_SR: SR;
	ESTOP_OK_TON: TON;
	ESTOP_ENA_ALM_TON: TON;	
	ESTOP_ALM_ENA_COMMON: BOOL;	
	OUTPUTS_SUPPLY_MAIN_GROUP_ENA: BOOL :=TRUE;	
	EStop_Healthy: BOOL;	
END_VAR

VAR_OUTPUT
	ESTOP_HEALHTY_COMMON: BOOL;	
END_VAR

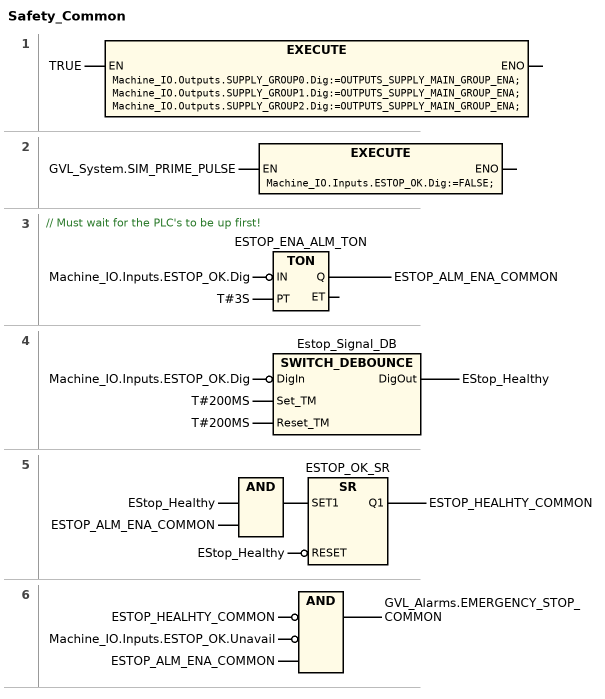
// NETWORK 1
Machine_IO.Outputs.SUPPLY_GROUP0.Dig:=OUTPUTS_SUPPLY_MAIN_GROUP_ENA;
Machine_IO.Outputs.SUPPLY_GROUP1.Dig:=OUTPUTS_SUPPLY_MAIN_GROUP_ENA;
Machine_IO.Outputs.SUPPLY_GROUP2.Dig:=OUTPUTS_SUPPLY_MAIN_GROUP_ENA;

// NETWORK 2
IF GVL_System.SIM_PRIME_PULSE THEN Machine_IO.Inputs.ESTOP_OK.Dig:=FALSE; END_IF

// NETWORK 3
// // Must wait for the PLC's to be up first!
ESTOP_ENA_ALM_TON(IN := NOT Machine_IO.Inputs.ESTOP_OK.Dig, PT := T#3S); // TON
ESTOP_ALM_ENA_COMMON := ESTOP_ENA_ALM_TON.Q;

// NETWORK 4
Estop_Signal_DB(DigIn := NOT Machine_IO.Inputs.ESTOP_OK.Dig, Set_TM := T#200MS, Reset_TM := T#200MS); // SWITCH_DEBOUNCE
EStop_Healthy := Estop_Signal_DB.DigOut;

// NETWORK 5
ESTOP_OK_SR(SET1 := EStop_Healthy AND ESTOP_ALM_ENA_COMMON, RESET := NOT EStop_Healthy); // SR
ESTOP_HEALHTY_COMMON := ESTOP_OK_SR.Q1;

// NETWORK 6
GVL_Alarms.EMERGENCY_STOP_COMMON := NOT ESTOP_HEALHTY_COMMON AND NOT Machine_IO.Inputs.ESTOP_OK.Unavail AND ESTOP_ALM_ENA_COMMON;

END_PROGRAM

// Device/Application/App_PLC/PLC_Alarms
PROGRAM PLC_Alarms
VAR
	LowOilPressureAlarm_TON: TON;
	EngineHighTempAlarm_TON: TON;
	LowHydOilAlarm_TON: TON;
	HydTempAlarm_TON: TON;
	LowFuelWarn_TON: ton;
	LowFuelAlarm_Set_TON: ton;
	LowFuelAlarm_Reset_TON: ton;
	DrumPressWarn_TON: ton;
	DrumPressureAlarm_TON: ton;
	FUEL_SYMBOL_DUTY: DUTY_CYCLE;
	Fuel_Symbol_Visible: BOOL;
END_VAR
VAR // added by the converter: edge detectors and wires of the graphical bodies
    _rt1 : R_TRIG;
    _w1 : BOOL;
END_VAR

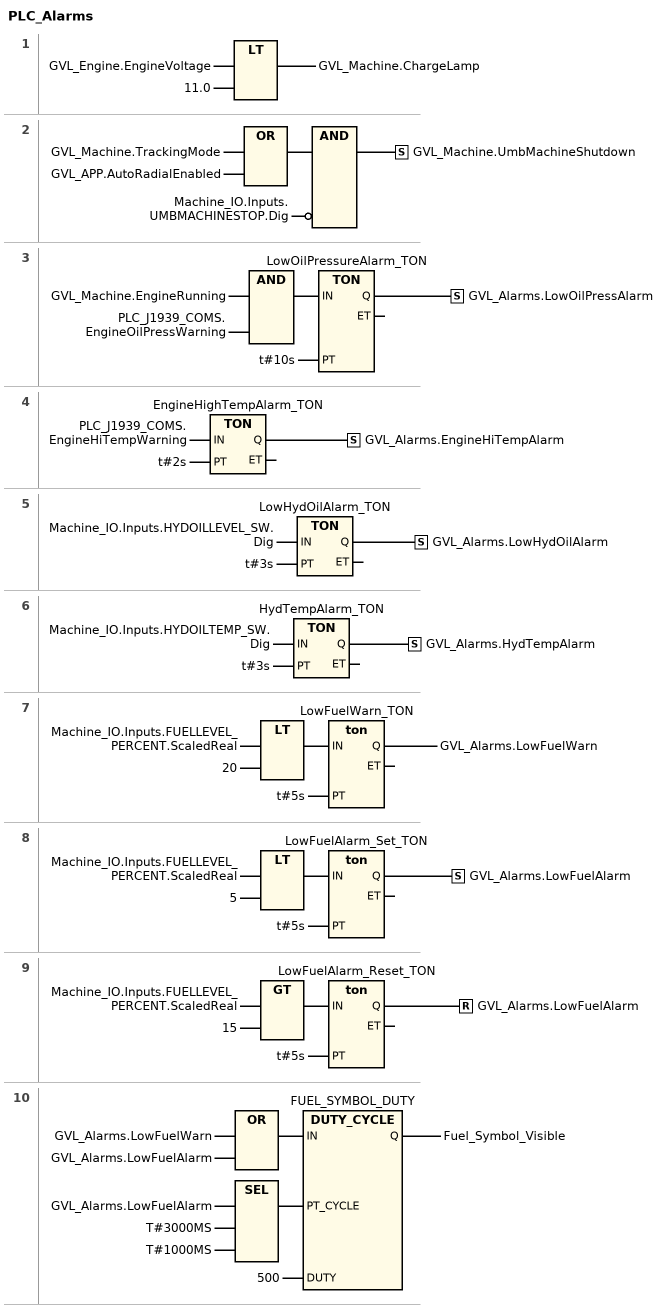
// NETWORK 1
GVL_Machine.ChargeLamp := GVL_Engine.EngineVoltage < 11.0;

// NETWORK 2
GVL_Machine.UmbMachineShutdown S= (GVL_Machine.TrackingMode OR GVL_APP.AutoRadialEnabled) AND NOT Machine_IO.Inputs.UMBMACHINESTOP.Dig;

// NETWORK 3
LowOilPressureAlarm_TON(IN := GVL_Machine.EngineRunning AND PLC_J1939_COMS.EngineOilPressWarning, PT := t#10s); // TON
GVL_Alarms.LowOilPressAlarm S= LowOilPressureAlarm_TON.Q;

// NETWORK 4
EngineHighTempAlarm_TON(IN := PLC_J1939_COMS.EngineHiTempWarning, PT := t#2s); // TON
GVL_Alarms.EngineHiTempAlarm S= EngineHighTempAlarm_TON.Q;

// NETWORK 5
LowHydOilAlarm_TON(IN := Machine_IO.Inputs.HYDOILLEVEL_SW.Dig, PT := t#3s); // TON
GVL_Alarms.LowHydOilAlarm S= LowHydOilAlarm_TON.Q;

// NETWORK 6
HydTempAlarm_TON(IN := Machine_IO.Inputs.HYDOILTEMP_SW.Dig, PT := t#3s); // TON
GVL_Alarms.HydTempAlarm S= HydTempAlarm_TON.Q;

// NETWORK 7
LowFuelWarn_TON(IN := Machine_IO.Inputs.FUELLEVEL_PERCENT.ScaledReal < 20, PT := t#5s); // ton
GVL_Alarms.LowFuelWarn := LowFuelWarn_TON.Q;

// NETWORK 8
LowFuelAlarm_Set_TON(IN := Machine_IO.Inputs.FUELLEVEL_PERCENT.ScaledReal < 5, PT := t#5s); // ton
GVL_Alarms.LowFuelAlarm S= LowFuelAlarm_Set_TON.Q;

// NETWORK 9
LowFuelAlarm_Reset_TON(IN := Machine_IO.Inputs.FUELLEVEL_PERCENT.ScaledReal > 15, PT := t#5s); // ton
GVL_Alarms.LowFuelAlarm R= LowFuelAlarm_Reset_TON.Q;

// NETWORK 10
FUEL_SYMBOL_DUTY(
    IN := GVL_Alarms.LowFuelWarn OR GVL_Alarms.LowFuelAlarm,
    PT_CYCLE := SEL(GVL_Alarms.LowFuelAlarm, T#3000MS, T#1000MS),
    DUTY := 500); // DUTY_CYCLE
Fuel_Symbol_Visible := FUEL_SYMBOL_DUTY.Q;

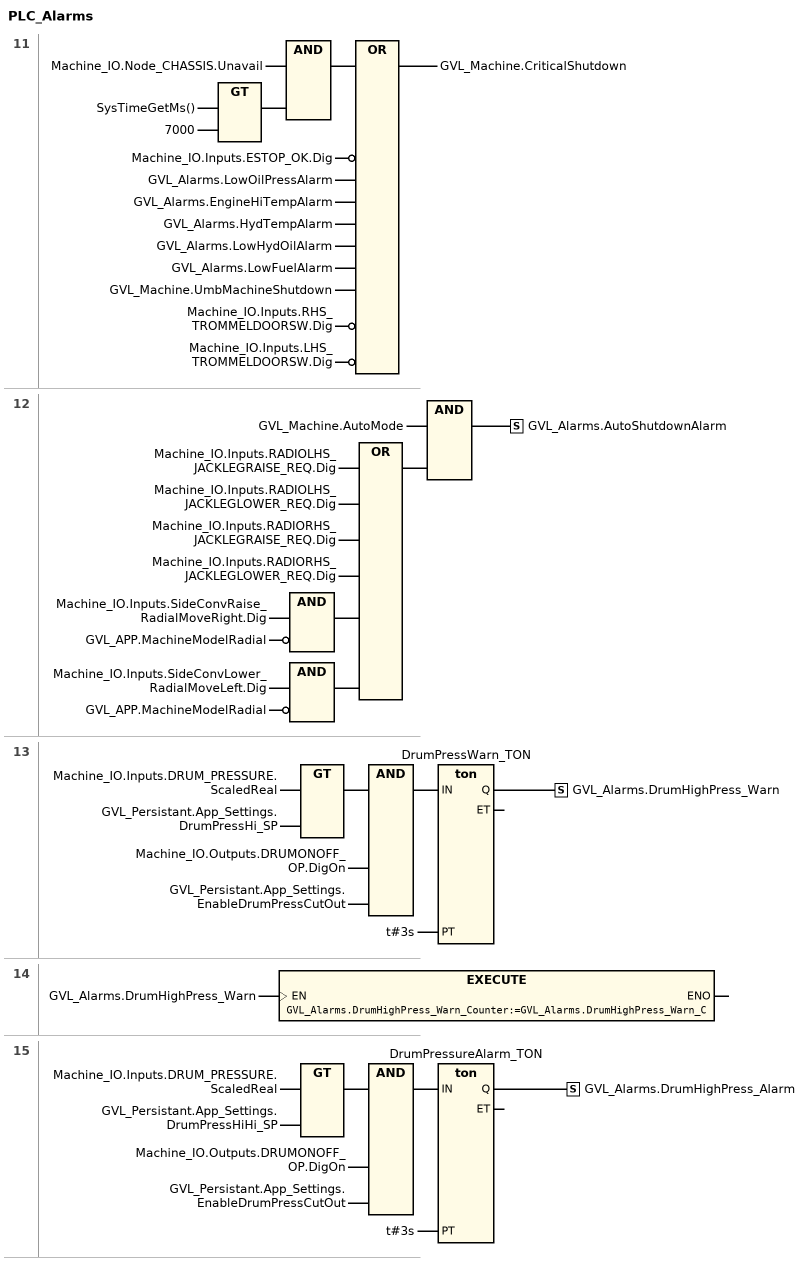
// NETWORK 11
GVL_Machine.CriticalShutdown := Machine_IO.Node_CHASSIS.Unavail AND (SysTimeGetMs()) > 7000 OR NOT Machine_IO.Inputs.ESTOP_OK.Dig OR GVL_Alarms.LowOilPressAlarm OR GVL_Alarms.EngineHiTempAlarm OR GVL_Alarms.HydTempAlarm OR GVL_Alarms.LowHydOilAlarm OR GVL_Alarms.LowFuelAlarm OR GVL_Machine.UmbMachineShutdown OR NOT Machine_IO.Inputs.RHS_TROMMELDOORSW.Dig OR NOT Machine_IO.Inputs.LHS_TROMMELDOORSW.Dig;

// NETWORK 12
GVL_Alarms.AutoShutdownAlarm S= GVL_Machine.AutoMode AND (Machine_IO.Inputs.RADIOLHS_JACKLEGRAISE_REQ.Dig OR Machine_IO.Inputs.RADIOLHS_JACKLEGLOWER_REQ.Dig OR Machine_IO.Inputs.RADIORHS_JACKLEGRAISE_REQ.Dig OR Machine_IO.Inputs.RADIORHS_JACKLEGLOWER_REQ.Dig OR Machine_IO.Inputs.SideConvRaise_RadialMoveRight.Dig AND NOT GVL_APP.MachineModelRadial OR Machine_IO.Inputs.SideConvLower_RadialMoveLeft.Dig AND NOT GVL_APP.MachineModelRadial);

// NETWORK 13
DrumPressWarn_TON(IN := Machine_IO.Inputs.DRUM_PRESSURE.ScaledReal > GVL_Persistant.App_Settings.DrumPressHi_SP AND Machine_IO.Outputs.DRUMONOFF_OP.DigOn AND GVL_Persistant.App_Settings.EnableDrumPressCutOut, PT := t#3s); // ton
GVL_Alarms.DrumHighPress_Warn S= DrumPressWarn_TON.Q;

// NETWORK 14
_rt1(CLK := GVL_Alarms.DrumHighPress_Warn);
IF _rt1.Q THEN GVL_Alarms.DrumHighPress_Warn_Counter:=GVL_Alarms.DrumHighPress_Warn_Counter+1; END_IF

// NETWORK 15
DrumPressureAlarm_TON(IN := Machine_IO.Inputs.DRUM_PRESSURE.ScaledReal > GVL_Persistant.App_Settings.DrumPressHiHi_SP AND Machine_IO.Outputs.DRUMONOFF_OP.DigOn AND GVL_Persistant.App_Settings.EnableDrumPressCutOut, PT := t#3s); // ton
GVL_Alarms.DrumHighPress_Alarm S= DrumPressureAlarm_TON.Q;

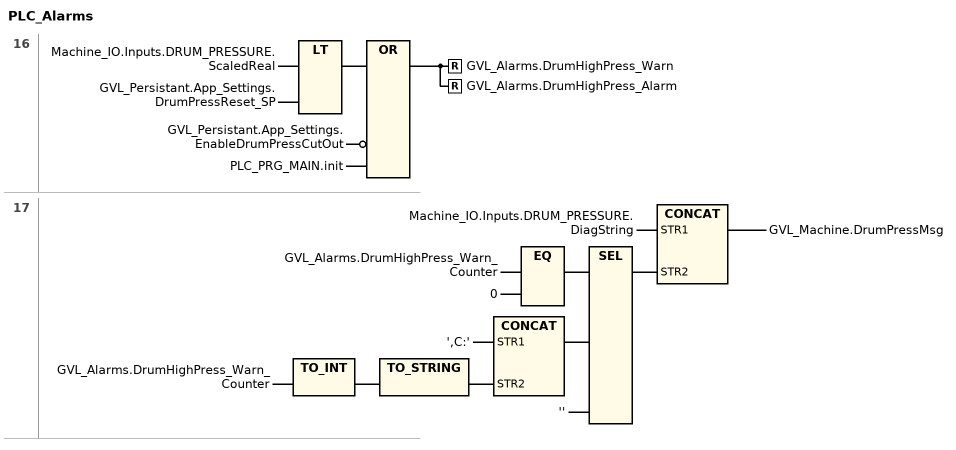
// NETWORK 16
_w1 := Machine_IO.Inputs.DRUM_PRESSURE.ScaledReal < GVL_Persistant.App_Settings.DrumPressReset_SP OR NOT GVL_Persistant.App_Settings.EnableDrumPressCutOut OR PLC_PRG_MAIN.init;
GVL_Alarms.DrumHighPress_Warn R= _w1;
GVL_Alarms.DrumHighPress_Alarm R= _w1;

// NETWORK 17
GVL_Machine.DrumPressMsg := CONCAT(STR1 := Machine_IO.Inputs.DRUM_PRESSURE.DiagString, STR2 := SEL(GVL_Alarms.DrumHighPress_Warn_Counter = 0, CONCAT(STR1 := ',C:', STR2 := TO_STRING(TO_INT(GVL_Alarms.DrumHighPress_Warn_Counter))), ''));

END_PROGRAM

// Device/Application/App_PLC/CAN Comms/Engine Comms/PLC_J1939_COMS
PROGRAM PLC_J1939_COMS
VAR
	Enable_CAN1: ifmRCAN.CAN_Enable;
	Status_CAN1: ifmRCAN.CAN_Status;
	
	ENA_J1939_DM1_DECODE: BOOL:=TRUE;
	ENA_J1939_TX_CUSTOM: BOOL:=TRUE;
	
	Coolant_Hi_Temp_DM1: PLC_DM1_Condition;
	EngineHiTempWarning: BOOL;
 	Engine_Oil_Press_Low_DM1: PLC_DM1_Condition;
	EngineOilPressWarning: BOOL;	
	DFP_LAMP_4_DUTY_CYCLE: DUTY_CYCLE;
	DFP_LAMP_2_DUTY_CYCLE: DUTY_CYCLE;
	SIM_DPF_Regen_Status: BOOL;
	Def_Duty_Flash: DUTY_CYCLE;
END_VAR

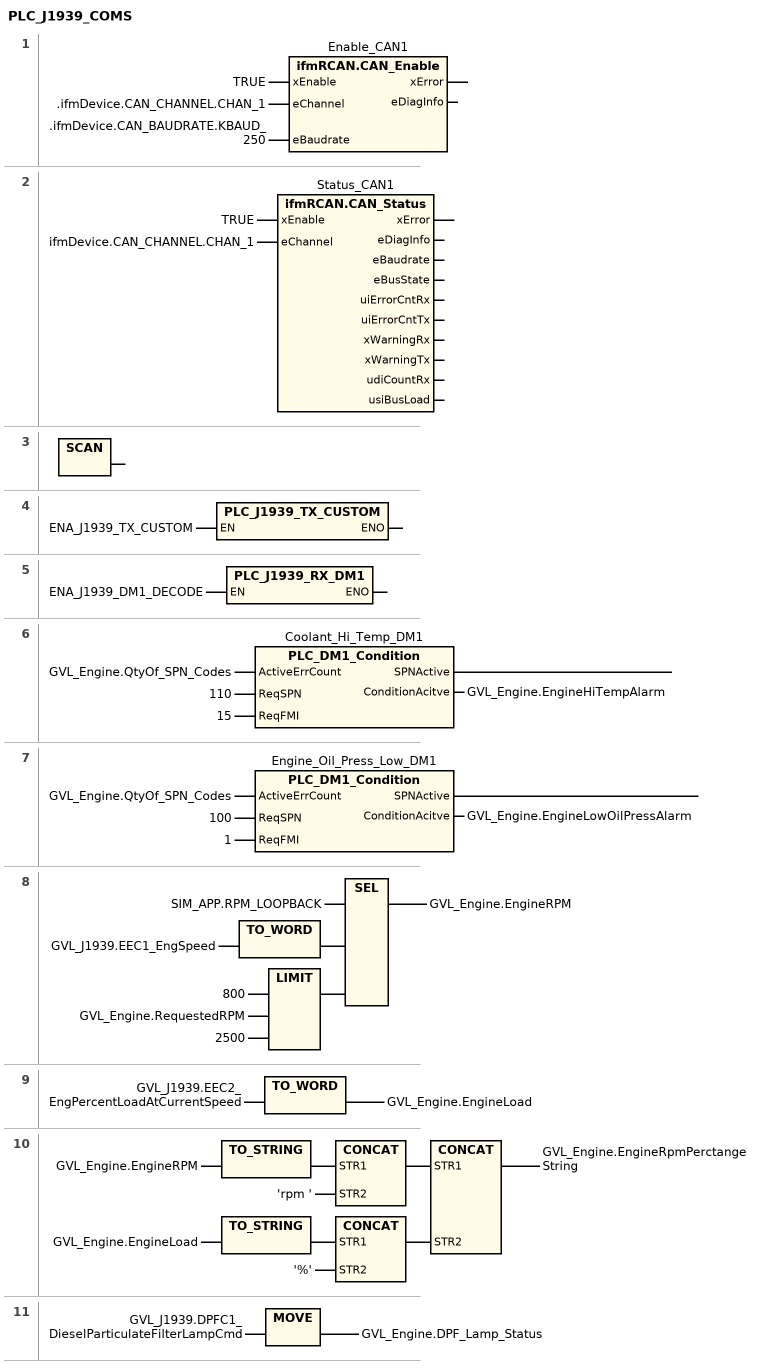
// NETWORK 1
Enable_CAN1(
    xEnable := TRUE,
    eChannel := .ifmDevice.CAN_CHANNEL.CHAN_1,
    eBaudrate := .ifmDevice.CAN_BAUDRATE.KBAUD_250); // ifmRCAN.CAN_Enable

// NETWORK 2
Status_CAN1(xEnable := TRUE, eChannel := ifmDevice.CAN_CHANNEL.CHAN_1); // ifmRCAN.CAN_Status

// NETWORK 3
SCAN();

// NETWORK 4
IF ENA_J1939_TX_CUSTOM THEN PLC_J1939_TX_CUSTOM(); END_IF

// NETWORK 5
IF ENA_J1939_DM1_DECODE THEN PLC_J1939_RX_DM1(); END_IF

// NETWORK 6
Coolant_Hi_Temp_DM1(
    ActiveErrCount := GVL_Engine.QtyOf_SPN_Codes,
    ReqSPN := 110,
    ReqFMI := 15,
    ConditionAcitve => GVL_Engine.EngineHiTempAlarm); // PLC_DM1_Condition

// NETWORK 7
Engine_Oil_Press_Low_DM1(
    ActiveErrCount := GVL_Engine.QtyOf_SPN_Codes,
    ReqSPN := 100,
    ReqFMI := 1,
    ConditionAcitve => GVL_Engine.EngineLowOilPressAlarm); // PLC_DM1_Condition

// NETWORK 8
GVL_Engine.EngineRPM := SEL(SIM_APP.RPM_LOOPBACK, TO_WORD(GVL_J1939.EEC1_EngSpeed), LIMIT(800, GVL_Engine.RequestedRPM, 2500));

// NETWORK 9
GVL_Engine.EngineLoad := TO_WORD(GVL_J1939.EEC2_EngPercentLoadAtCurrentSpeed);

// NETWORK 10
GVL_Engine.EngineRpmPerctangeString := CONCAT(STR1 := CONCAT(STR1 := TO_STRING(GVL_Engine.EngineRPM), STR2 := 'rpm '), STR2 := CONCAT(STR1 := TO_STRING(GVL_Engine.EngineLoad), STR2 := '%'));

// NETWORK 11
GVL_Engine.DPF_Lamp_Status := GVL_J1939.DPFC1_DieselParticulateFilterLampCmd;

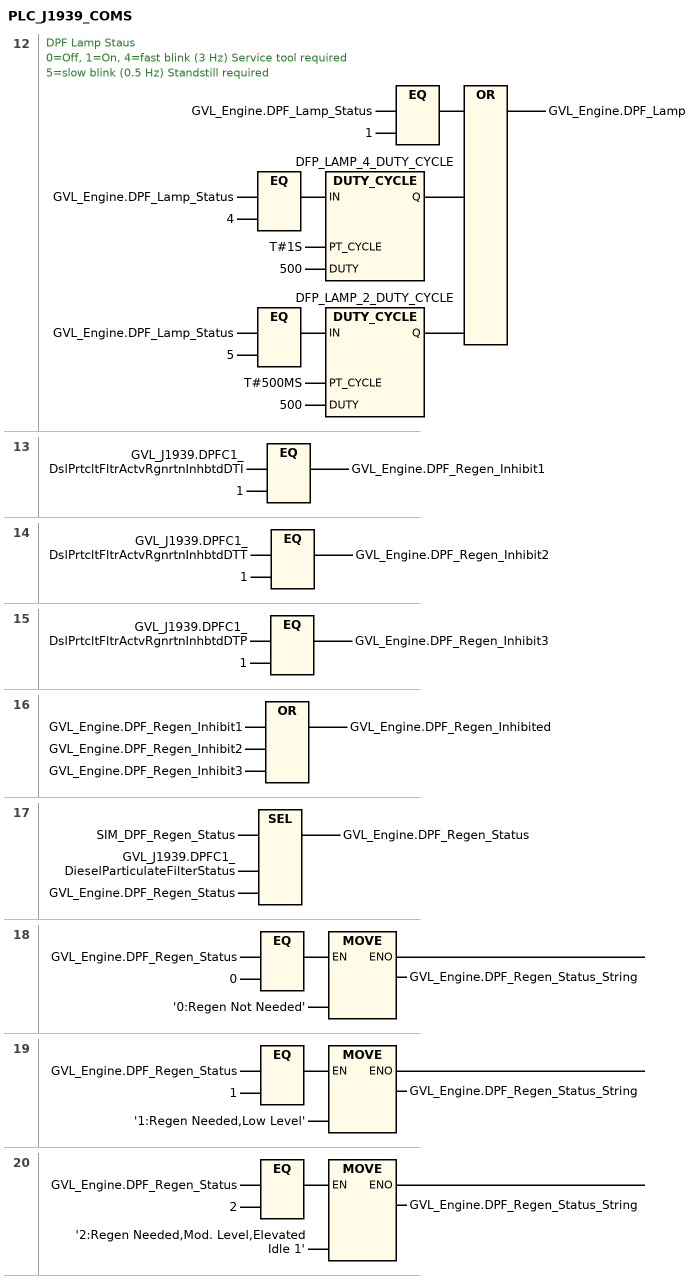
// NETWORK 12
// DPF Lamp Staus
// 0=Off, 1=On, 4=fast blink (3 Hz) Service tool required
// 5=slow blink (0.5 Hz) Standstill required
DFP_LAMP_4_DUTY_CYCLE(IN := GVL_Engine.DPF_Lamp_Status = 4, PT_CYCLE := T#1S, DUTY := 500); // DUTY_CYCLE
DFP_LAMP_2_DUTY_CYCLE(IN := GVL_Engine.DPF_Lamp_Status = 5, PT_CYCLE := T#500MS, DUTY := 500); // DUTY_CYCLE
GVL_Engine.DPF_Lamp := GVL_Engine.DPF_Lamp_Status = 1 OR DFP_LAMP_4_DUTY_CYCLE.Q OR DFP_LAMP_2_DUTY_CYCLE.Q;

// NETWORK 13
GVL_Engine.DPF_Regen_Inhibit1 := GVL_J1939.DPFC1_DslPrtcltFltrActvRgnrtnInhbtdDTI = 1;

// NETWORK 14
GVL_Engine.DPF_Regen_Inhibit2 := GVL_J1939.DPFC1_DslPrtcltFltrActvRgnrtnInhbtdDTT = 1;

// NETWORK 15
GVL_Engine.DPF_Regen_Inhibit3 := GVL_J1939.DPFC1_DslPrtcltFltrActvRgnrtnInhbtdDTP = 1;

// NETWORK 16
GVL_Engine.DPF_Regen_Inhibited := GVL_Engine.DPF_Regen_Inhibit1 OR GVL_Engine.DPF_Regen_Inhibit2 OR GVL_Engine.DPF_Regen_Inhibit3;

// NETWORK 17
GVL_Engine.DPF_Regen_Status := SEL(SIM_DPF_Regen_Status, GVL_J1939.DPFC1_DieselParticulateFilterStatus, GVL_Engine.DPF_Regen_Status);

// NETWORK 18
IF GVL_Engine.DPF_Regen_Status = 0 THEN GVL_Engine.DPF_Regen_Status_String := '0:Regen Not Needed'; END_IF

// NETWORK 19
IF GVL_Engine.DPF_Regen_Status = 1 THEN GVL_Engine.DPF_Regen_Status_String := '1:Regen Needed,Low Level'; END_IF

// NETWORK 20
IF GVL_Engine.DPF_Regen_Status = 2 THEN
    GVL_Engine.DPF_Regen_Status_String := '2:Regen Needed,Mod. Level,Elevated Idle 1';
END_IF

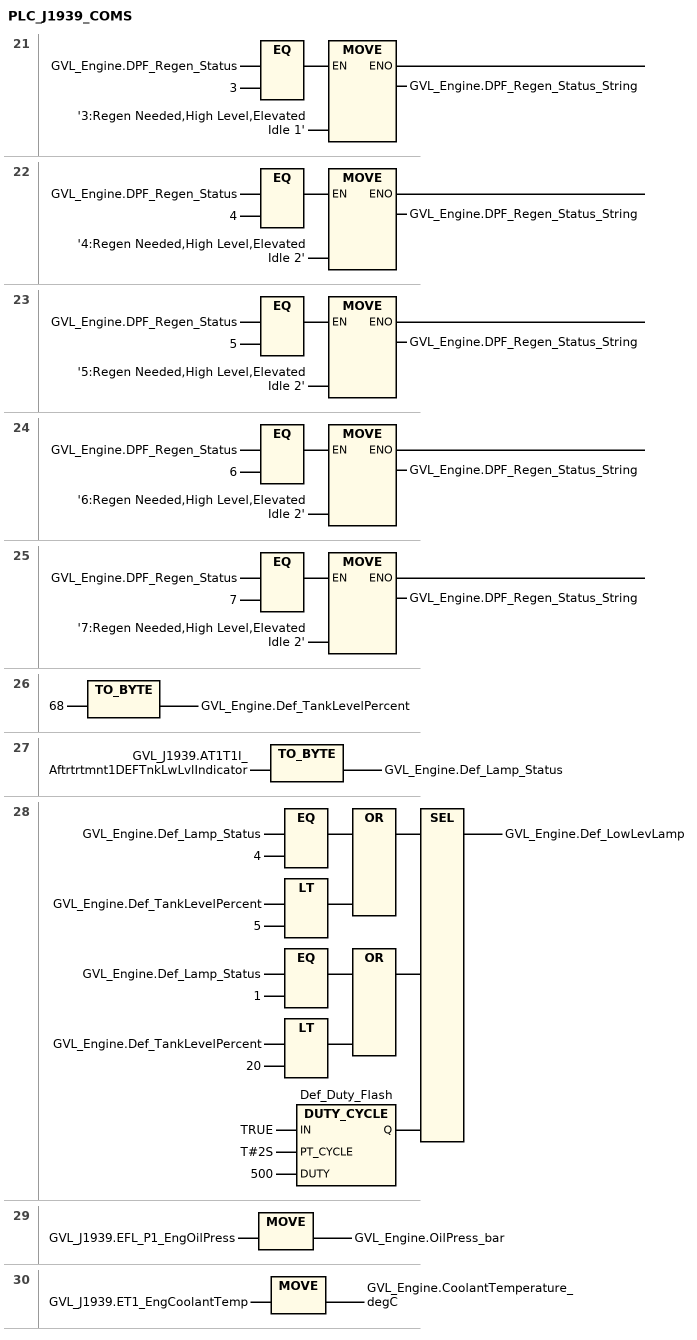
// NETWORK 21
IF GVL_Engine.DPF_Regen_Status = 3 THEN
    GVL_Engine.DPF_Regen_Status_String := '3:Regen Needed,High Level,Elevated Idle 1';
END_IF

// NETWORK 22
IF GVL_Engine.DPF_Regen_Status = 4 THEN
    GVL_Engine.DPF_Regen_Status_String := '4:Regen Needed,High Level,Elevated Idle 2';
END_IF

// NETWORK 23
IF GVL_Engine.DPF_Regen_Status = 5 THEN
    GVL_Engine.DPF_Regen_Status_String := '5:Regen Needed,High Level,Elevated Idle 2';
END_IF

// NETWORK 24
IF GVL_Engine.DPF_Regen_Status = 6 THEN
    GVL_Engine.DPF_Regen_Status_String := '6:Regen Needed,High Level,Elevated Idle 2';
END_IF

// NETWORK 25
IF GVL_Engine.DPF_Regen_Status = 7 THEN
    GVL_Engine.DPF_Regen_Status_String := '7:Regen Needed,High Level,Elevated Idle 2';
END_IF

// NETWORK 26
GVL_Engine.Def_TankLevelPercent := TO_BYTE(68);

// NETWORK 27
GVL_Engine.Def_Lamp_Status := TO_BYTE(GVL_J1939.AT1T1I_Aftrtrtmnt1DEFTnkLwLvlIndicator);

// NETWORK 28
Def_Duty_Flash(IN := TRUE, PT_CYCLE := T#2S, DUTY := 500); // DUTY_CYCLE
GVL_Engine.Def_LowLevLamp := SEL(GVL_Engine.Def_Lamp_Status = 4 OR GVL_Engine.Def_TankLevelPercent < 5, GVL_Engine.Def_Lamp_Status = 1 OR GVL_Engine.Def_TankLevelPercent < 20, Def_Duty_Flash.Q);

// NETWORK 29
GVL_Engine.OilPress_bar := GVL_J1939.EFL_P1_EngOilPress;

// NETWORK 30
GVL_Engine.CoolantTemperature_degC := GVL_J1939.ET1_EngCoolantTemp;

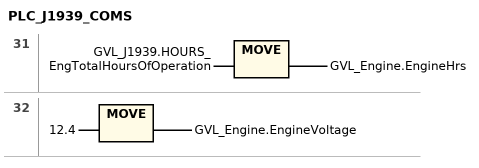
// NETWORK 31
GVL_Engine.EngineHrs := GVL_J1939.HOURS_EngTotalHoursOfOperation;

// NETWORK 32
GVL_Engine.EngineVoltage := 12.4;

METHOD SCAN
VAR_INPUT
END_VAR
GVL_J1939.EEC1_ActualEngPercentTorque;
GVL_J1939.EEC1_EngSpeed;
GVL_J1939.EEC2_EngPercentLoadAtCurrentSpeed;
GVL_J1939.EEC2_SCRThermalManagementActive;
GVL_J1939.EEC2_ActlMxAvailableEngPercentTorque;
GVL_J1939.EEC3_NominalFrictionPercentTorque;
GVL_J1939.EEC3_EngsDesiredOperatingSpeed;
GVL_J1939.EEC5_EngExhstGsRcrculation1ValveCtrl;
GVL_J1939.ET1_EngCoolantTemp;
GVL_J1939.ET1_EngFuelTemp1;
GVL_J1939.EFL_P1_EngOilPress;
GVL_J1939.EFL_P1_EngCoolantLevel;
GVL_J1939.EFL_P2_EngInjectorMeteringRail1Press;
GVL_J1939.LFC_EngTotalFuelUsed;
GVL_J1939.AMB_BarometricPress;
GVL_J1939.AMB_AmbientAirTemp;
GVL_J1939.AMB_EngAirIntakeTemp;
GVL_J1939.IC1_EngIntakeManifold1Press;
GVL_J1939.IC1_EngIntakeManifold1Temp;
GVL_J1939.IC1_EngAirIntakePress;
GVL_J1939.VEP1_BatteryPotential_PowerInput1;
GVL_J1939.VEP1_KeyswitchBatteryPotential;
GVL_J1939.EFS_EngOilPrimingState;
GVL_J1939.EFS_FuelPumpPrimerStatus;
GVL_J1939.DPFC1_DieselParticulateFilterLampCmd;
GVL_J1939.DPFC1_DslPrtcltFltrActvRgnrtionStatus;
GVL_J1939.DPFC1_DieselParticulateFilterStatus;
GVL_J1939.DPFC1_DslPrtcltFltrActvRgnrtnInhbtdDTI;
GVL_J1939.DPFC1_DslPrtcltFltrActvRgnrtnInhbtdDTT;
GVL_J1939.DPFC1_DslPrtcltFltrActvRgnrtnInhbtdDTP;
GVL_J1939.AT1IG2_Aftrtrtmnt1DslPrtcltFltrInt_0000;
GVL_J1939.AT1T1I_Aftrtrtmnt1SCRCatalystTankLevel;
GVL_J1939.AT1T1I_Aftrtrtment1SCRCatalystTankTemp;
GVL_J1939.AT1T1I_Aftrtrtmnt1DEFTnkLwLvlIndicator;
GVL_J1939.AT1T1I_AftrtrtmntSCROprtrIndcmntSvrity;
GVL_J1939.A1SCRDSI1_Aftertreatment1SCRSystemState;
GVL_J1939.A1SCREGT_Aftrtrtmnt1SCRCtlystIntkGasTemp;
GVL_J1939.A1DOC_Aftrtrtmnt1DslOxdtnCtlystIn_0000;
GVL_J1939.WFI_WaterInFuelIndicator;
GVL_J1939.DLCC1_EngAirFilterRestrictionLampCmd;
GVL_J1939.DLCD1_EngOilPressLowLampData;
GVL_J1939.DLCD1_EngCoolantLevelLowLampData;
END_METHOD

END_PROGRAM

// Device/Application/App_PLC/CAN Comms/Engine Comms/PLC_J1939_TX_CUSTOM
PROGRAM PLC_J1939_TX_CUSTOM
VAR
	Tx_TSC1: ifmrcan.CAN_Tx;
	TSC1_Ton1: TON;
	
	Standstill_RegenRelease: BOOL;
	RegenInhibit: BOOL:=FALSE;
	
	Tx_CM1: ifmrcan.CAN_Tx;
	CM1_Ton1: TON;
	Tx_CM2: ifmrcan.CAN_Tx;
	CM2_Ton1: TON;

	ElevateRpmAllowed_PBTog: PIL.PB_Toggle;
	TSC1_CheckSum: CounterChecksum;
	TSC1_WTB_12: PIL.WordToByte;

	HOURS_Request_Payload: ARRAY [0..7] OF USINT := [16#E5,16#FE,0,0,0,0,0,0];	
	HOURS_Request_PGN_CAN_Tx: ifmrcan.CAN_Tx;
	HOURS_Request_TON: TON;
	
	TX_TSC1_Error_Counter: WORD;
END_VAR

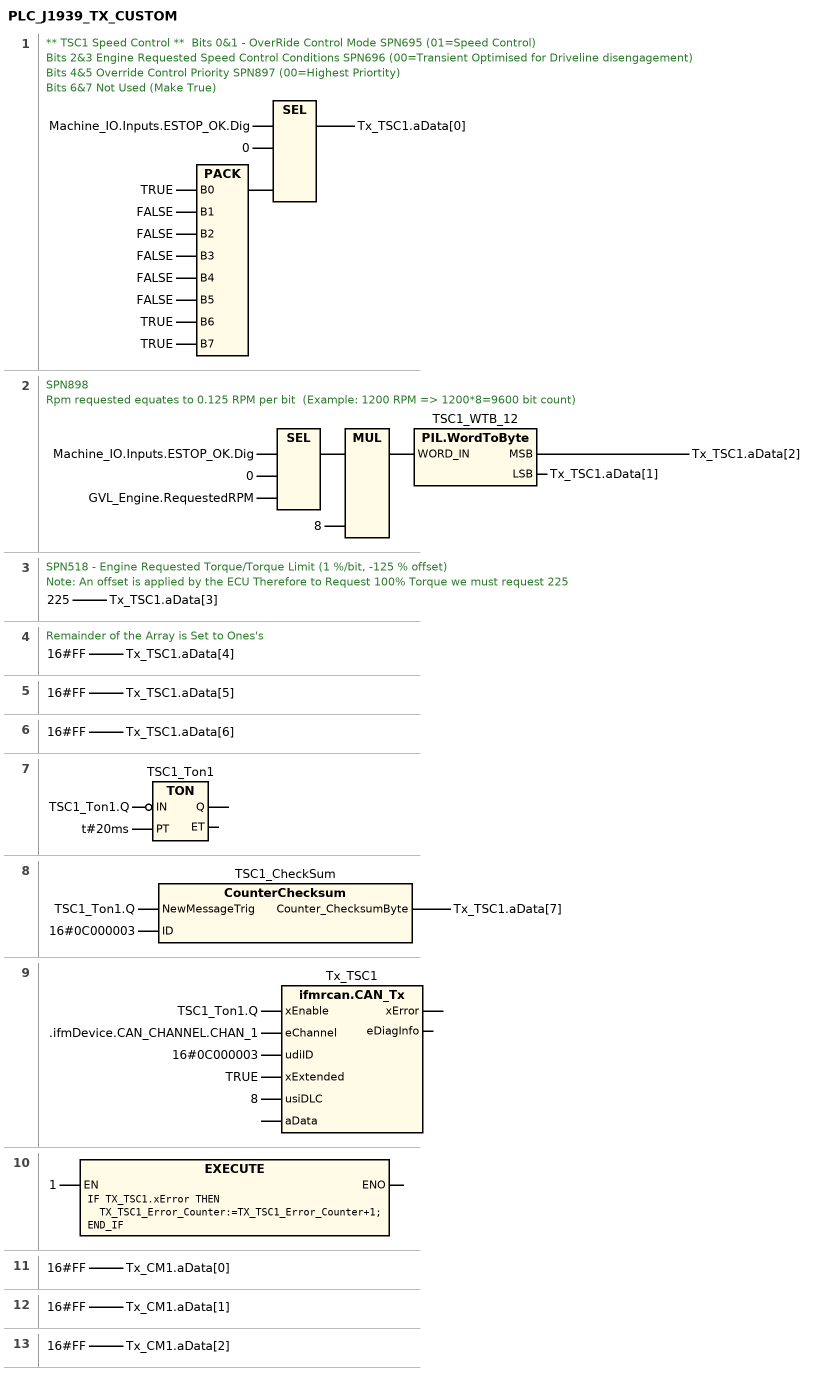
// NETWORK 1
// 					** TSC1 Speed Control **  Bits 0&1 - OverRide Control Mode SPN695 (01=Speed Control)
// Bits 2&3 Engine Requested Speed Control Conditions SPN696 (00=Transient Optimised for Driveline disengagement)
// Bits 4&5 Override Control Priority SPN897 (00=Highest Priortity)
// Bits 6&7 Not Used (Make True)
//
Tx_TSC1.aData[0] := SEL(Machine_IO.Inputs.ESTOP_OK.Dig, 0, PACK(B0 := TRUE, B1 := FALSE, B2 := FALSE, B3 := FALSE, B4 := FALSE, B5 := FALSE, B6 := TRUE, B7 := TRUE));

// NETWORK 2
// 					SPN898
// Rpm requested equates to 0.125 RPM per bit  (Example: 1200 RPM => 1200*8=9600 bit count)
//
TSC1_WTB_12(WORD_IN := SEL(Machine_IO.Inputs.ESTOP_OK.Dig, 0, GVL_Engine.RequestedRPM) * 8, LSB => Tx_TSC1.aData[1]); // PIL.WordToByte
Tx_TSC1.aData[2] := TSC1_WTB_12.MSB;

// NETWORK 3
// 					SPN518 - Engine Requested Torque/Torque Limit (1 %/bit, -125 % offset)
// Note: An offset is applied by the ECU Therefore to Request 100% Torque we must request 225
//
Tx_TSC1.aData[3] := 225;

// NETWORK 4
// Remainder of the Array is Set to Ones's
Tx_TSC1.aData[4] := 16#FF;

// NETWORK 5
Tx_TSC1.aData[5] := 16#FF;

// NETWORK 6
Tx_TSC1.aData[6] := 16#FF;

// NETWORK 7
TSC1_Ton1(IN := NOT TSC1_Ton1.Q, PT := t#20ms); // TON

// NETWORK 8
TSC1_CheckSum(NewMessageTrig := TSC1_Ton1.Q, ID := 16#0C000003); // CounterChecksum
Tx_TSC1.aData[7] := TSC1_CheckSum.Counter_ChecksumByte;

// NETWORK 9
Tx_TSC1(
    xEnable := TSC1_Ton1.Q,
    eChannel := .ifmDevice.CAN_CHANNEL.CHAN_1,
    udiID := 16#0C000003,
    xExtended := TRUE,
    usiDLC := 8); // ifmrcan.CAN_Tx

// NETWORK 10
IF 1 THEN
    IF TX_TSC1.xError THEN
    	TX_TSC1_Error_Counter:=TX_TSC1_Error_Counter+1;
    END_IF
END_IF

// NETWORK 11
Tx_CM1.aData[0] := 16#FF;

// NETWORK 12
Tx_CM1.aData[1] := 16#FF;

// NETWORK 13
Tx_CM1.aData[2] := 16#FF;

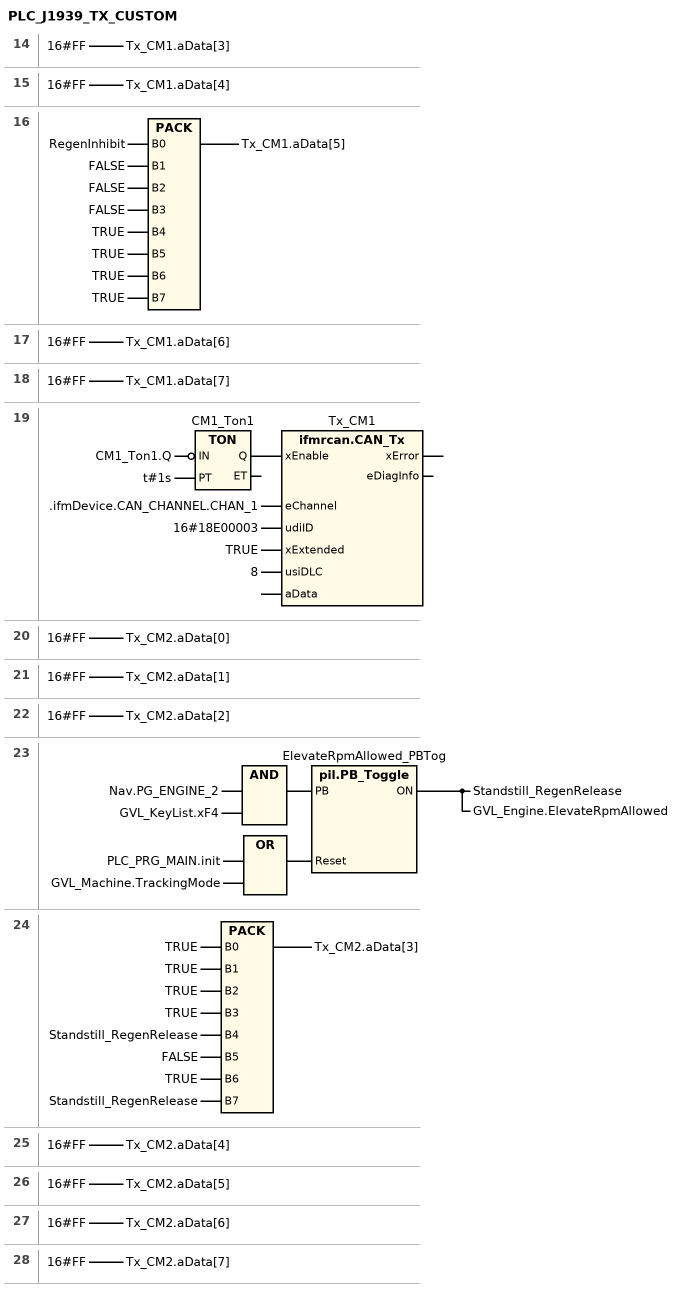
// NETWORK 14
Tx_CM1.aData[3] := 16#FF;

// NETWORK 15
Tx_CM1.aData[4] := 16#FF;

// NETWORK 16
Tx_CM1.aData[5] := PACK(B0 := RegenInhibit, B1 := FALSE, B2 := FALSE, B3 := FALSE, B4 := TRUE, B5 := TRUE, B6 := TRUE, B7 := TRUE);

// NETWORK 17
Tx_CM1.aData[6] := 16#FF;

// NETWORK 18
Tx_CM1.aData[7] := 16#FF;

// NETWORK 19
CM1_Ton1(IN := NOT CM1_Ton1.Q, PT := t#1s); // TON
Tx_CM1(
    xEnable := CM1_Ton1.Q,
    eChannel := .ifmDevice.CAN_CHANNEL.CHAN_1,
    udiID := 16#18E00003,
    xExtended := TRUE,
    usiDLC := 8); // ifmrcan.CAN_Tx

// NETWORK 20
Tx_CM2.aData[0] := 16#FF;

// NETWORK 21
Tx_CM2.aData[1] := 16#FF;

// NETWORK 22
Tx_CM2.aData[2] := 16#FF;

// NETWORK 23
ElevateRpmAllowed_PBTog(PB := Nav.PG_ENGINE_2 AND GVL_KeyList.xF4, Reset := PLC_PRG_MAIN.init OR GVL_Machine.TrackingMode); // pil.PB_Toggle
Standstill_RegenRelease := ElevateRpmAllowed_PBTog.ON;
GVL_Engine.ElevateRpmAllowed := ElevateRpmAllowed_PBTog.ON;

// NETWORK 24
Tx_CM2.aData[3] := PACK(B0 := TRUE, B1 := TRUE, B2 := TRUE, B3 := TRUE, B4 := Standstill_RegenRelease, B5 := FALSE, B6 := TRUE, B7 := Standstill_RegenRelease);

// NETWORK 25
Tx_CM2.aData[4] := 16#FF;

// NETWORK 26
Tx_CM2.aData[5] := 16#FF;

// NETWORK 27
Tx_CM2.aData[6] := 16#FF;

// NETWORK 28
Tx_CM2.aData[7] := 16#FF;

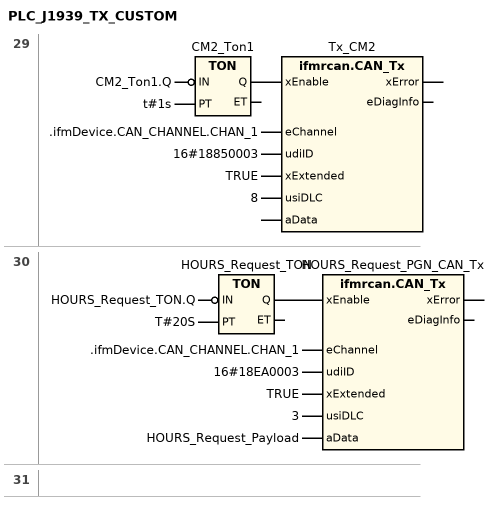
// NETWORK 29
CM2_Ton1(IN := NOT CM2_Ton1.Q, PT := t#1s); // TON
Tx_CM2(
    xEnable := CM2_Ton1.Q,
    eChannel := .ifmDevice.CAN_CHANNEL.CHAN_1,
    udiID := 16#18850003,
    xExtended := TRUE,
    usiDLC := 8); // ifmrcan.CAN_Tx

// NETWORK 30
HOURS_Request_TON(IN := NOT HOURS_Request_TON.Q, PT := T#20S); // TON
HOURS_Request_PGN_CAN_Tx(
    xEnable := HOURS_Request_TON.Q,
    eChannel := .ifmDevice.CAN_CHANNEL.CHAN_1,
    udiID := 16#18EA0003,
    xExtended := TRUE,
    usiDLC := 3,
    aData := HOURS_Request_Payload); // ifmrcan.CAN_Tx

// NETWORK 31

END_PROGRAM

// Device/Application/App_PLC/CAN Comms/Engine Comms/CounterChecksum
FUNCTION_BLOCK CounterChecksum
VAR
	MessageCounter: BYTE;
	CheckSum: DWORD;
	MessageCheckSum: BYTE;
	ID_Low: BYTE;
	ID_midLow: BYTE;
	ID_midHigh: BYTE;
	ID_High: BYTE;
END_VAR
VAR_INPUT
	NewMessageTrig: BOOL;
	ID: DWORD;
END_VAR
VAR_OUTPUT
	Counter_ChecksumByte: BYTE;
END_VAR

ID_Low:=DWORD_TO_BYTE(ID);
ID_midLow:=DWORD_TO_BYTE(SHR(ID,8));
ID_midHigh:=DWORD_TO_BYTE(SHR(ID,16));
ID_High:=DWORD_TO_BYTE(SHR(ID,24));


IF NewMessageTrig=TRUE THEN MessageCounter:=MessageCounter+1;END_IF
IF MessageCounter>7 THEN MessageCounter:=0; END_IF

CheckSum:=PLC_J1939_TX_CUSTOM.Tx_TSC1.aData[0]+PLC_J1939_TX_CUSTOM.Tx_TSC1.aData[1]+PLC_J1939_TX_CUSTOM.Tx_TSC1.aData[2]+PLC_J1939_TX_CUSTOM.Tx_TSC1.aData[3]+
				PLC_J1939_TX_CUSTOM.Tx_TSC1.aData[4]+PLC_J1939_TX_CUSTOM.Tx_TSC1.aData[5]+PLC_J1939_TX_CUSTOM.Tx_TSC1.aData[6]+(MessageCounter AND 16#0F) + ID_Low + ID_midLow + ID_midHigh + ID_High;

MessageCheckSum:= DWORD_TO_BYTE((((SHR(CheckSum,6)) AND 16#03)+(SHR(CheckSum,3))+CheckSum) AND 16#07);

Counter_ChecksumByte:=SHL(MessageCheckSum,4)+MessageCounter;

END_FUNCTION_BLOCK

// Device/Application/App_PLC/CAN Comms/Engine Comms/PLC_J1939_RX_DM1
PROGRAM PLC_J1939_RX_DM1
VAR
	DM1_Index_Count: CTUD;
	DM1_Rx_FECA: ifmrcan.CAN_Rx;

	P2Bits_EngineProtectLamp: Pack2bits;
	P2Bits_EngineWarningLamp: Pack2bits;
	P2Bits_EngineStopLamp: Pack2bits;
	P2Bits_MILamp: Pack2bits;

	SPN_Code: DWORD;
	FMI_Code: BYTE;
	OC_Code: BYTE;

	DM1_FECA_Data: ARRAY [0..7] OF USINT;
	DM1_ECFF_Data: ARRAY [0..7] OF USINT;
	BAM_EBFF_Data: ARRAY [0..7] OF USINT;

	BAM_Rx_ECFF: ifmrcan.CAN_Rx;
	BAM_ECFF_RxFlag: BOOL;
	BtDw_BAM_DM1: PIL.ByteToDword;
	BAM_NumberOfBytes: INT;
	BtW_NumberOfBytes: PIL.ByteToWord;
	BAM_DM1: BOOL;
	BAM_Rx_EBFF: ifmrcan.CAN_Rx;
	EBFF_RxFlag: BOOL;
	LampStatus: BYTE;
	DM1_Array: ARRAY [0..32] OF BYTE;
	
	Extract_SPN_1: fb_Extract_SPN;
	Extract_SPN_2: fb_Extract_SPN;
	Extract_SPN_3: fb_Extract_SPN;
	Extract_SPN_4: fb_Extract_SPN;
	Extract_SPN_5: fb_Extract_SPN;
	Extract_SPN_6: fb_Extract_SPN;
	Extract_SPN_7: fb_Extract_SPN;
	Extract_SPN_8: fb_Extract_SPN;
	
	SPN_Array: ARRAY [1..8] OF DWORD;
	FMI_Array: ARRAY [1..8] OF BYTE;
	OC_Array: ARRAY [1..8] OF BYTE;

	DM1_FECA_Rec: BOOL;
	DM1_BAM_No_Of_Packets: BYTE;
	DM1_BAM_Packet_Count: CTU;
END_VAR
VAR // added by the converter: edge detectors and wires of the graphical bodies
    _w1, _w2, _w3 : BOOL;
END_VAR

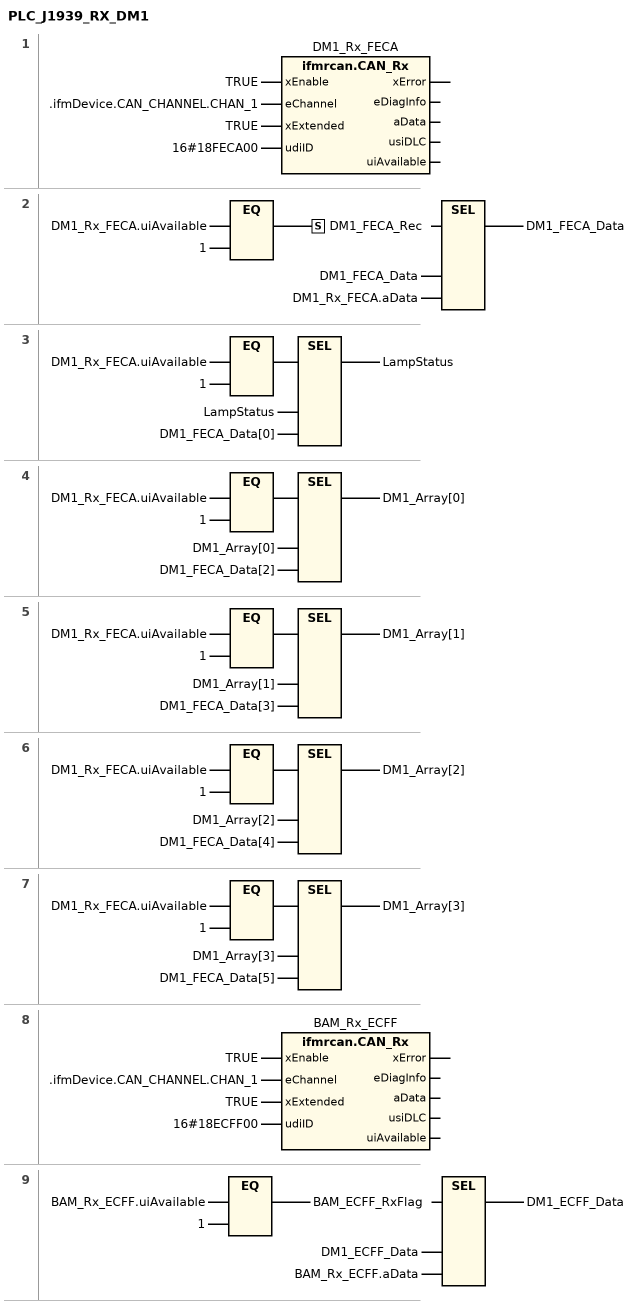
// NETWORK 1
DM1_Rx_FECA(
    xEnable := TRUE,
    eChannel := .ifmDevice.CAN_CHANNEL.CHAN_1,
    xExtended := TRUE,
    udiID := 16#18FECA00); // ifmrcan.CAN_Rx

// NETWORK 2
_w1 := DM1_Rx_FECA.uiAvailable = 1;
DM1_FECA_Rec S= _w1;
DM1_FECA_Data := SEL(_w1, DM1_FECA_Data, DM1_Rx_FECA.aData);

// NETWORK 3
LampStatus := SEL(DM1_Rx_FECA.uiAvailable = 1, LampStatus, DM1_FECA_Data[0]);

// NETWORK 4
DM1_Array[0] := SEL(DM1_Rx_FECA.uiAvailable = 1, DM1_Array[0], DM1_FECA_Data[2]);

// NETWORK 5
DM1_Array[1] := SEL(DM1_Rx_FECA.uiAvailable = 1, DM1_Array[1], DM1_FECA_Data[3]);

// NETWORK 6
DM1_Array[2] := SEL(DM1_Rx_FECA.uiAvailable = 1, DM1_Array[2], DM1_FECA_Data[4]);

// NETWORK 7
DM1_Array[3] := SEL(DM1_Rx_FECA.uiAvailable = 1, DM1_Array[3], DM1_FECA_Data[5]);

// NETWORK 8
BAM_Rx_ECFF(
    xEnable := TRUE,
    eChannel := .ifmDevice.CAN_CHANNEL.CHAN_1,
    xExtended := TRUE,
    udiID := 16#18ECFF00); // ifmrcan.CAN_Rx

// NETWORK 9
_w2 := BAM_Rx_ECFF.uiAvailable = 1;
BAM_ECFF_RxFlag := _w2;
DM1_ECFF_Data := SEL(_w2, DM1_ECFF_Data, BAM_Rx_ECFF.aData);

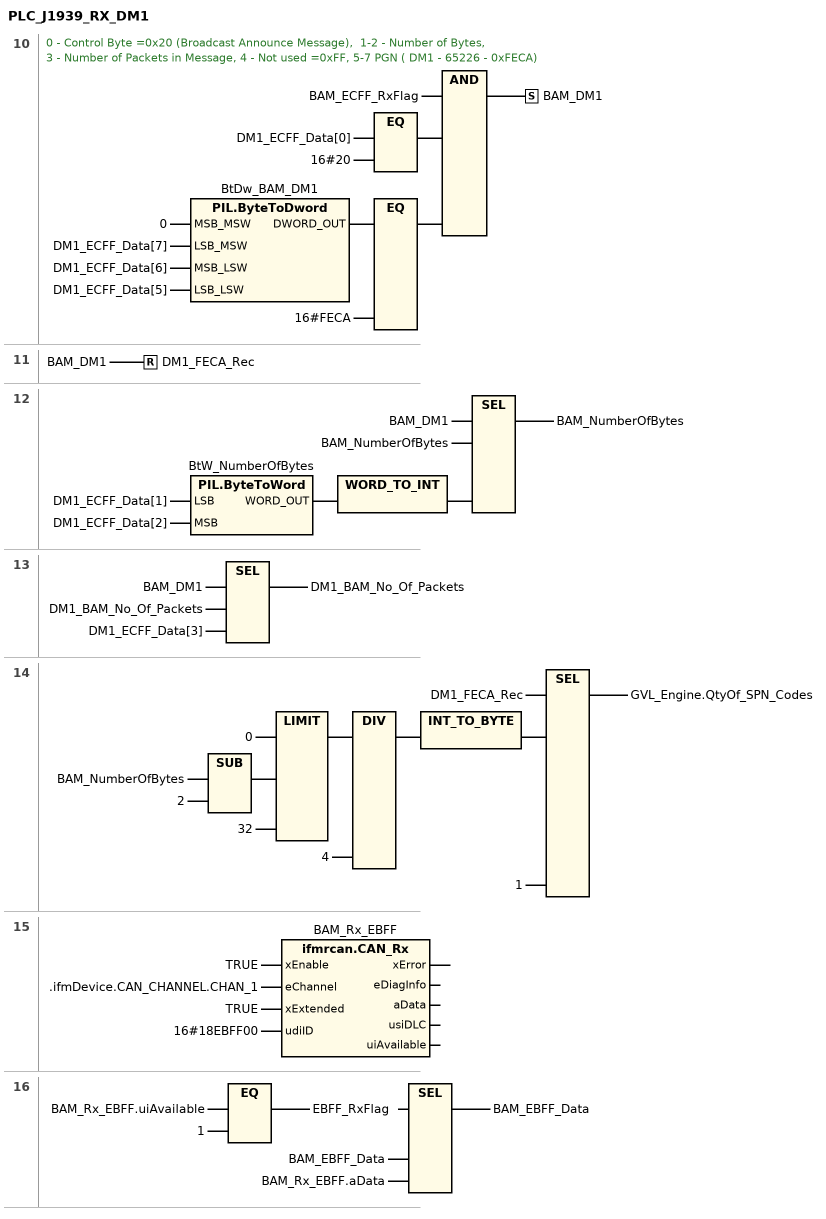
// NETWORK 10
// 					0 - Control Byte =0x20 (Broadcast Announce Message),  1-2 - Number of Bytes,
// 3 - Number of Packets in Message, 4 - Not used =0xFF, 5-7 PGN ( DM1 - 65226 - 0xFECA)
//
BtDw_BAM_DM1(
    MSB_MSW := 0,
    LSB_MSW := DM1_ECFF_Data[7],
    MSB_LSW := DM1_ECFF_Data[6],
    LSB_LSW := DM1_ECFF_Data[5]); // PIL.ByteToDword
BAM_DM1 S= BAM_ECFF_RxFlag AND DM1_ECFF_Data[0] = 16#20 AND BtDw_BAM_DM1.DWORD_OUT = 16#FECA;

// NETWORK 11
DM1_FECA_Rec R= BAM_DM1;

// NETWORK 12
BtW_NumberOfBytes(LSB := DM1_ECFF_Data[1], MSB := DM1_ECFF_Data[2]); // PIL.ByteToWord
BAM_NumberOfBytes := SEL(BAM_DM1, BAM_NumberOfBytes, WORD_TO_INT(BtW_NumberOfBytes.WORD_OUT));

// NETWORK 13
DM1_BAM_No_Of_Packets := SEL(BAM_DM1, DM1_BAM_No_Of_Packets, DM1_ECFF_Data[3]);

// NETWORK 14
GVL_Engine.QtyOf_SPN_Codes := SEL(DM1_FECA_Rec, INT_TO_BYTE(LIMIT(0, BAM_NumberOfBytes - 2, 32) / 4), 1);

// NETWORK 15
BAM_Rx_EBFF(
    xEnable := TRUE,
    eChannel := .ifmDevice.CAN_CHANNEL.CHAN_1,
    xExtended := TRUE,
    udiID := 16#18EBFF00); // ifmrcan.CAN_Rx

// NETWORK 16
_w3 := BAM_Rx_EBFF.uiAvailable = 1;
EBFF_RxFlag := _w3;
BAM_EBFF_Data := SEL(_w3, BAM_EBFF_Data, BAM_Rx_EBFF.aData);

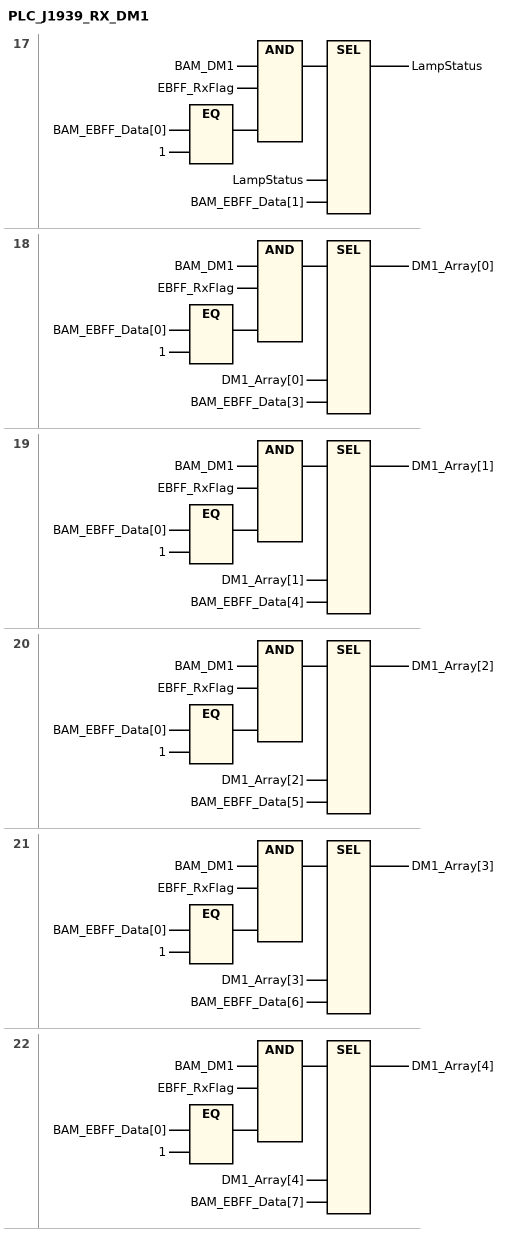
// NETWORK 17
LampStatus := SEL(BAM_DM1 AND EBFF_RxFlag AND BAM_EBFF_Data[0] = 1, LampStatus, BAM_EBFF_Data[1]);

// NETWORK 18
DM1_Array[0] := SEL(BAM_DM1 AND EBFF_RxFlag AND BAM_EBFF_Data[0] = 1, DM1_Array[0], BAM_EBFF_Data[3]);

// NETWORK 19
DM1_Array[1] := SEL(BAM_DM1 AND EBFF_RxFlag AND BAM_EBFF_Data[0] = 1, DM1_Array[1], BAM_EBFF_Data[4]);

// NETWORK 20
DM1_Array[2] := SEL(BAM_DM1 AND EBFF_RxFlag AND BAM_EBFF_Data[0] = 1, DM1_Array[2], BAM_EBFF_Data[5]);

// NETWORK 21
DM1_Array[3] := SEL(BAM_DM1 AND EBFF_RxFlag AND BAM_EBFF_Data[0] = 1, DM1_Array[3], BAM_EBFF_Data[6]);

// NETWORK 22
DM1_Array[4] := SEL(BAM_DM1 AND EBFF_RxFlag AND BAM_EBFF_Data[0] = 1, DM1_Array[4], BAM_EBFF_Data[7]);

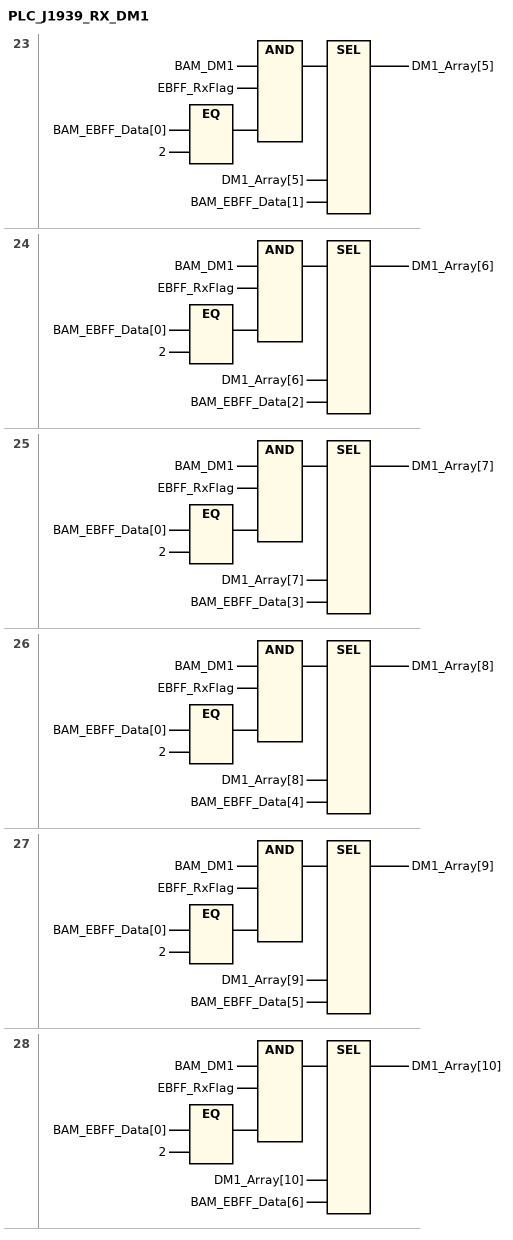
// NETWORK 23
DM1_Array[5] := SEL(BAM_DM1 AND EBFF_RxFlag AND BAM_EBFF_Data[0] = 2, DM1_Array[5], BAM_EBFF_Data[1]);

// NETWORK 24
DM1_Array[6] := SEL(BAM_DM1 AND EBFF_RxFlag AND BAM_EBFF_Data[0] = 2, DM1_Array[6], BAM_EBFF_Data[2]);

// NETWORK 25
DM1_Array[7] := SEL(BAM_DM1 AND EBFF_RxFlag AND BAM_EBFF_Data[0] = 2, DM1_Array[7], BAM_EBFF_Data[3]);

// NETWORK 26
DM1_Array[8] := SEL(BAM_DM1 AND EBFF_RxFlag AND BAM_EBFF_Data[0] = 2, DM1_Array[8], BAM_EBFF_Data[4]);

// NETWORK 27
DM1_Array[9] := SEL(BAM_DM1 AND EBFF_RxFlag AND BAM_EBFF_Data[0] = 2, DM1_Array[9], BAM_EBFF_Data[5]);

// NETWORK 28
DM1_Array[10] := SEL(BAM_DM1 AND EBFF_RxFlag AND BAM_EBFF_Data[0] = 2, DM1_Array[10], BAM_EBFF_Data[6]);

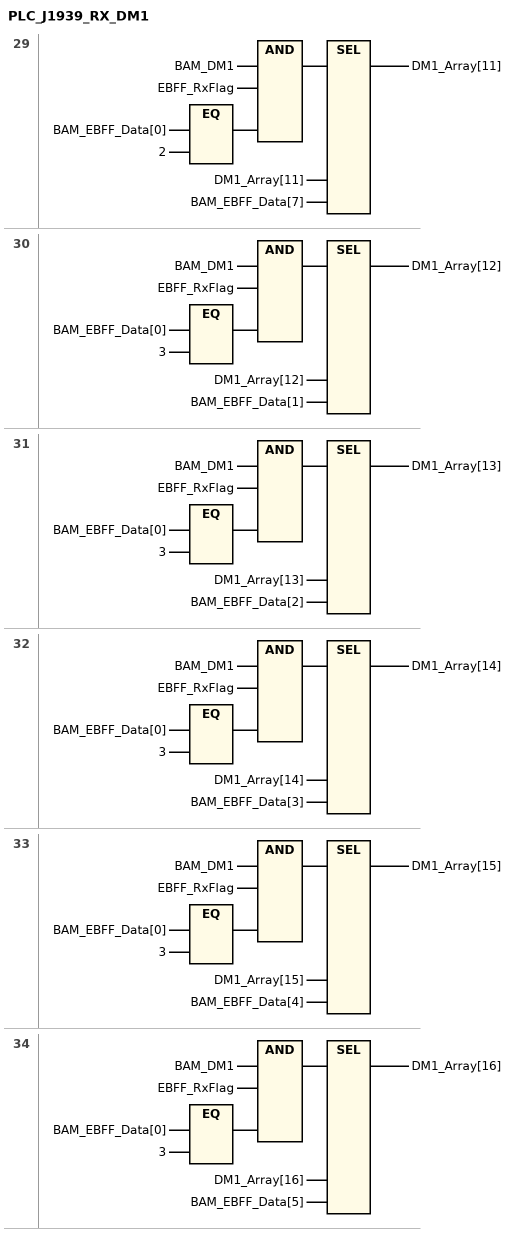
// NETWORK 29
DM1_Array[11] := SEL(BAM_DM1 AND EBFF_RxFlag AND BAM_EBFF_Data[0] = 2, DM1_Array[11], BAM_EBFF_Data[7]);

// NETWORK 30
DM1_Array[12] := SEL(BAM_DM1 AND EBFF_RxFlag AND BAM_EBFF_Data[0] = 3, DM1_Array[12], BAM_EBFF_Data[1]);

// NETWORK 31
DM1_Array[13] := SEL(BAM_DM1 AND EBFF_RxFlag AND BAM_EBFF_Data[0] = 3, DM1_Array[13], BAM_EBFF_Data[2]);

// NETWORK 32
DM1_Array[14] := SEL(BAM_DM1 AND EBFF_RxFlag AND BAM_EBFF_Data[0] = 3, DM1_Array[14], BAM_EBFF_Data[3]);

// NETWORK 33
DM1_Array[15] := SEL(BAM_DM1 AND EBFF_RxFlag AND BAM_EBFF_Data[0] = 3, DM1_Array[15], BAM_EBFF_Data[4]);

// NETWORK 34
DM1_Array[16] := SEL(BAM_DM1 AND EBFF_RxFlag AND BAM_EBFF_Data[0] = 3, DM1_Array[16], BAM_EBFF_Data[5]);

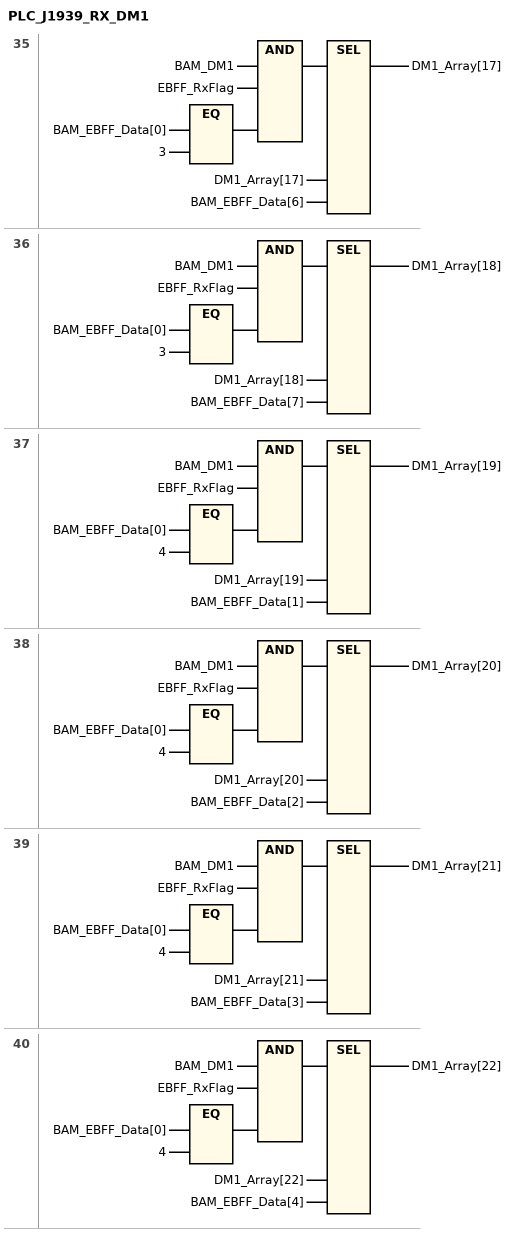
// NETWORK 35
DM1_Array[17] := SEL(BAM_DM1 AND EBFF_RxFlag AND BAM_EBFF_Data[0] = 3, DM1_Array[17], BAM_EBFF_Data[6]);

// NETWORK 36
DM1_Array[18] := SEL(BAM_DM1 AND EBFF_RxFlag AND BAM_EBFF_Data[0] = 3, DM1_Array[18], BAM_EBFF_Data[7]);

// NETWORK 37
DM1_Array[19] := SEL(BAM_DM1 AND EBFF_RxFlag AND BAM_EBFF_Data[0] = 4, DM1_Array[19], BAM_EBFF_Data[1]);

// NETWORK 38
DM1_Array[20] := SEL(BAM_DM1 AND EBFF_RxFlag AND BAM_EBFF_Data[0] = 4, DM1_Array[20], BAM_EBFF_Data[2]);

// NETWORK 39
DM1_Array[21] := SEL(BAM_DM1 AND EBFF_RxFlag AND BAM_EBFF_Data[0] = 4, DM1_Array[21], BAM_EBFF_Data[3]);

// NETWORK 40
DM1_Array[22] := SEL(BAM_DM1 AND EBFF_RxFlag AND BAM_EBFF_Data[0] = 4, DM1_Array[22], BAM_EBFF_Data[4]);

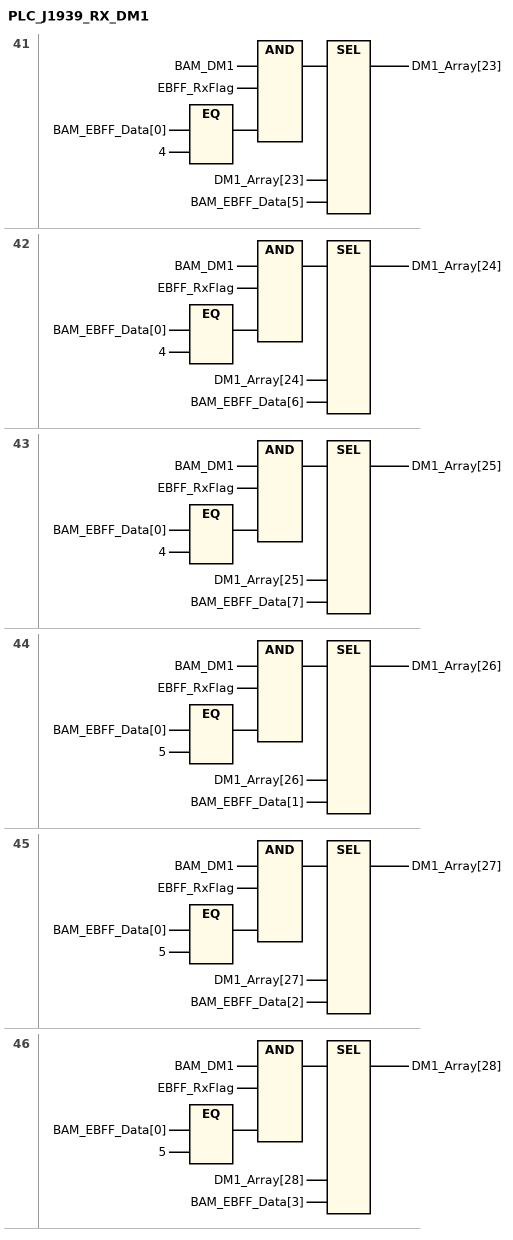
// NETWORK 41
DM1_Array[23] := SEL(BAM_DM1 AND EBFF_RxFlag AND BAM_EBFF_Data[0] = 4, DM1_Array[23], BAM_EBFF_Data[5]);

// NETWORK 42
DM1_Array[24] := SEL(BAM_DM1 AND EBFF_RxFlag AND BAM_EBFF_Data[0] = 4, DM1_Array[24], BAM_EBFF_Data[6]);

// NETWORK 43
DM1_Array[25] := SEL(BAM_DM1 AND EBFF_RxFlag AND BAM_EBFF_Data[0] = 4, DM1_Array[25], BAM_EBFF_Data[7]);

// NETWORK 44
DM1_Array[26] := SEL(BAM_DM1 AND EBFF_RxFlag AND BAM_EBFF_Data[0] = 5, DM1_Array[26], BAM_EBFF_Data[1]);

// NETWORK 45
DM1_Array[27] := SEL(BAM_DM1 AND EBFF_RxFlag AND BAM_EBFF_Data[0] = 5, DM1_Array[27], BAM_EBFF_Data[2]);

// NETWORK 46
DM1_Array[28] := SEL(BAM_DM1 AND EBFF_RxFlag AND BAM_EBFF_Data[0] = 5, DM1_Array[28], BAM_EBFF_Data[3]);

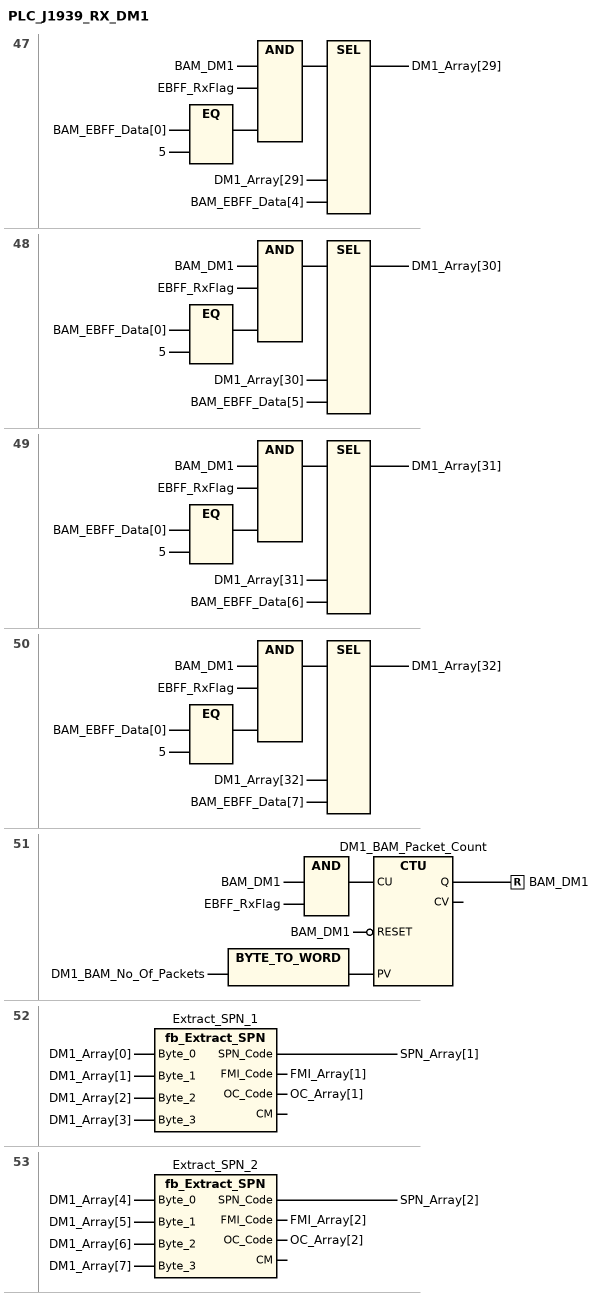
// NETWORK 47
DM1_Array[29] := SEL(BAM_DM1 AND EBFF_RxFlag AND BAM_EBFF_Data[0] = 5, DM1_Array[29], BAM_EBFF_Data[4]);

// NETWORK 48
DM1_Array[30] := SEL(BAM_DM1 AND EBFF_RxFlag AND BAM_EBFF_Data[0] = 5, DM1_Array[30], BAM_EBFF_Data[5]);

// NETWORK 49
DM1_Array[31] := SEL(BAM_DM1 AND EBFF_RxFlag AND BAM_EBFF_Data[0] = 5, DM1_Array[31], BAM_EBFF_Data[6]);

// NETWORK 50
DM1_Array[32] := SEL(BAM_DM1 AND EBFF_RxFlag AND BAM_EBFF_Data[0] = 5, DM1_Array[32], BAM_EBFF_Data[7]);

// NETWORK 51
DM1_BAM_Packet_Count(
    CU := BAM_DM1 AND EBFF_RxFlag,
    RESET := NOT BAM_DM1,
    PV := BYTE_TO_WORD(DM1_BAM_No_Of_Packets)); // CTU
BAM_DM1 R= DM1_BAM_Packet_Count.Q;

// NETWORK 52
Extract_SPN_1(
    Byte_0 := DM1_Array[0],
    Byte_1 := DM1_Array[1],
    Byte_2 := DM1_Array[2],
    Byte_3 := DM1_Array[3],
    FMI_Code => FMI_Array[1],
    OC_Code => OC_Array[1]); // fb_Extract_SPN
SPN_Array[1] := Extract_SPN_1.SPN_Code;

// NETWORK 53
Extract_SPN_2(
    Byte_0 := DM1_Array[4],
    Byte_1 := DM1_Array[5],
    Byte_2 := DM1_Array[6],
    Byte_3 := DM1_Array[7],
    FMI_Code => FMI_Array[2],
    OC_Code => OC_Array[2]); // fb_Extract_SPN
SPN_Array[2] := Extract_SPN_2.SPN_Code;

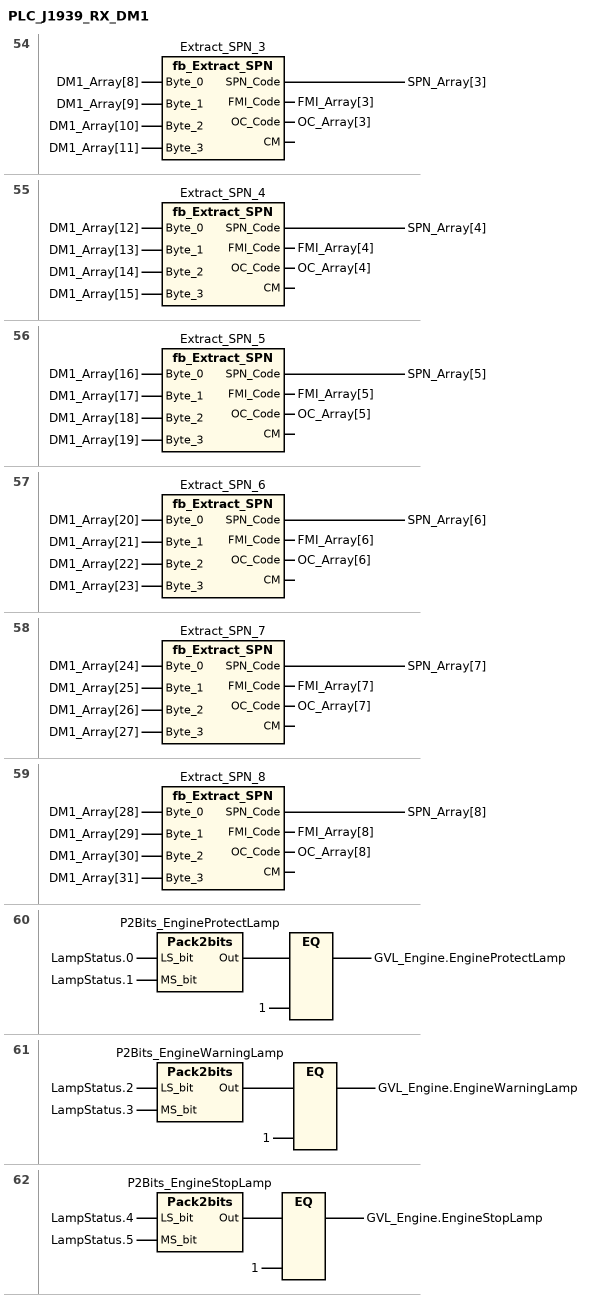
// NETWORK 54
Extract_SPN_3(
    Byte_0 := DM1_Array[8],
    Byte_1 := DM1_Array[9],
    Byte_2 := DM1_Array[10],
    Byte_3 := DM1_Array[11],
    FMI_Code => FMI_Array[3],
    OC_Code => OC_Array[3]); // fb_Extract_SPN
SPN_Array[3] := Extract_SPN_3.SPN_Code;

// NETWORK 55
Extract_SPN_4(
    Byte_0 := DM1_Array[12],
    Byte_1 := DM1_Array[13],
    Byte_2 := DM1_Array[14],
    Byte_3 := DM1_Array[15],
    FMI_Code => FMI_Array[4],
    OC_Code => OC_Array[4]); // fb_Extract_SPN
SPN_Array[4] := Extract_SPN_4.SPN_Code;

// NETWORK 56
Extract_SPN_5(
    Byte_0 := DM1_Array[16],
    Byte_1 := DM1_Array[17],
    Byte_2 := DM1_Array[18],
    Byte_3 := DM1_Array[19],
    FMI_Code => FMI_Array[5],
    OC_Code => OC_Array[5]); // fb_Extract_SPN
SPN_Array[5] := Extract_SPN_5.SPN_Code;

// NETWORK 57
Extract_SPN_6(
    Byte_0 := DM1_Array[20],
    Byte_1 := DM1_Array[21],
    Byte_2 := DM1_Array[22],
    Byte_3 := DM1_Array[23],
    FMI_Code => FMI_Array[6],
    OC_Code => OC_Array[6]); // fb_Extract_SPN
SPN_Array[6] := Extract_SPN_6.SPN_Code;

// NETWORK 58
Extract_SPN_7(
    Byte_0 := DM1_Array[24],
    Byte_1 := DM1_Array[25],
    Byte_2 := DM1_Array[26],
    Byte_3 := DM1_Array[27],
    FMI_Code => FMI_Array[7],
    OC_Code => OC_Array[7]); // fb_Extract_SPN
SPN_Array[7] := Extract_SPN_7.SPN_Code;

// NETWORK 59
Extract_SPN_8(
    Byte_0 := DM1_Array[28],
    Byte_1 := DM1_Array[29],
    Byte_2 := DM1_Array[30],
    Byte_3 := DM1_Array[31],
    FMI_Code => FMI_Array[8],
    OC_Code => OC_Array[8]); // fb_Extract_SPN
SPN_Array[8] := Extract_SPN_8.SPN_Code;

// NETWORK 60
P2Bits_EngineProtectLamp(LS_bit := LampStatus.0, MS_bit := LampStatus.1); // Pack2bits
GVL_Engine.EngineProtectLamp := P2Bits_EngineProtectLamp.Out = 1;

// NETWORK 61
P2Bits_EngineWarningLamp(LS_bit := LampStatus.2, MS_bit := LampStatus.3); // Pack2bits
GVL_Engine.EngineWarningLamp := P2Bits_EngineWarningLamp.Out = 1;

// NETWORK 62
P2Bits_EngineStopLamp(LS_bit := LampStatus.4, MS_bit := LampStatus.5); // Pack2bits
GVL_Engine.EngineStopLamp := P2Bits_EngineStopLamp.Out = 1;

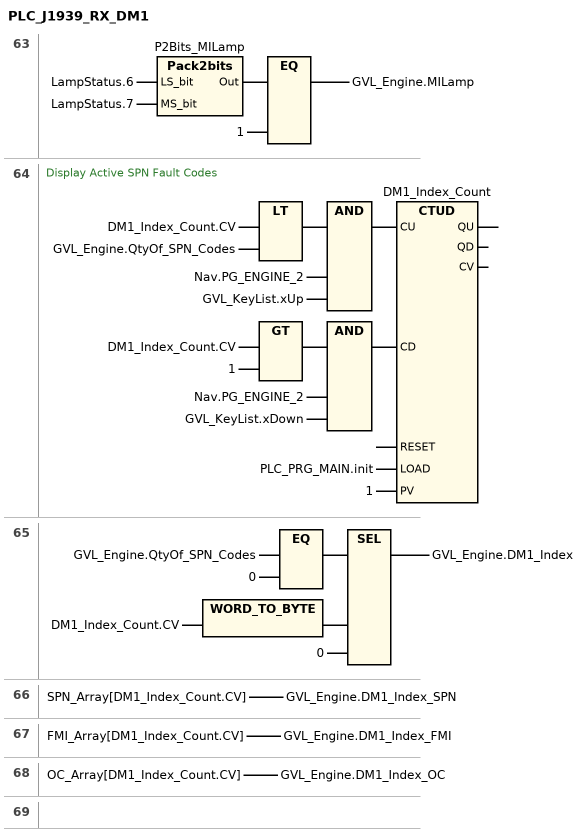
// NETWORK 63
P2Bits_MILamp(LS_bit := LampStatus.6, MS_bit := LampStatus.7); // Pack2bits
GVL_Engine.MILamp := P2Bits_MILamp.Out = 1;

// NETWORK 64
// Display Active SPN Fault Codes
DM1_Index_Count(
    CU := DM1_Index_Count.CV < GVL_Engine.QtyOf_SPN_Codes AND Nav.PG_ENGINE_2 AND GVL_KeyList.xUp,
    CD := DM1_Index_Count.CV > 1 AND Nav.PG_ENGINE_2 AND GVL_KeyList.xDown,
    LOAD := PLC_PRG_MAIN.init,
    PV := 1); // CTUD

// NETWORK 65
GVL_Engine.DM1_Index := SEL(GVL_Engine.QtyOf_SPN_Codes = 0, WORD_TO_BYTE(DM1_Index_Count.CV), 0);

// NETWORK 66
GVL_Engine.DM1_Index_SPN := SPN_Array[DM1_Index_Count.CV];

// NETWORK 67
GVL_Engine.DM1_Index_FMI := FMI_Array[DM1_Index_Count.CV];

// NETWORK 68
GVL_Engine.DM1_Index_OC := OC_Array[DM1_Index_Count.CV];

// NETWORK 69

END_PROGRAM

// Device/Application/App_PLC/CAN Comms/Engine Comms/fb_Extract_SPN
FUNCTION_BLOCK fb_Extract_SPN
VAR
	BtDW1: PIL.ByteToDword;
END_VAR
VAR_INPUT
	Byte_0: BYTE;
	Byte_1: BYTE;
	Byte_2: BYTE;
	Byte_3: BYTE;
END_VAR
VAR_OUTPUT
	SPN_Code: DWORD;
	FMI_Code: BYTE;
	OC_Code: BYTE;
	CM: BOOL;
END_VAR

